(* PLC project PhysicsSimulator, Nammo OpenPLC 1 *)
(* stored: creationDateTime 2026-02-23T12:09:45, modificationDateTime 2026-02-23T12:09:45 *)

TYPE TANK_T : STRUCT
  tank_id : INT;
  status : INT;
  x_position : REAL;
  y_position : REAL;
  z_position : REAL;
  stn_type : INT;
END_STRUCT;
END_TYPE

TYPE STATION_T : STRUCT
  tank_id : INT;
  status : INT;
  x_position : REAL;
  y_position : REAL;
  z_position : REAL;
  stn_type : INT;
  dropping_time : REAL;
  device_delay : REAL;
END_STRUCT;
END_TYPE

TYPE PHYSICS_2D_T : STRUCT
  x_accel_s : REAL;
  x_decel_s : REAL;
  x_max_mm_s : REAL;
  z_total_mm : REAL;
  z_slow_dry_mm : REAL;
  z_slow_wet_mm : REAL;
  z_slow_end_mm : REAL;
  z_slow_mm_s : REAL;
  z_fast_mm_s : REAL;
  drip_delay_s : REAL;
  avoid_mm : REAL;
END_STRUCT;
END_TYPE

TYPE TASK_AREA_T : STRUCT
  min_lift : INT;
  max_lift : INT;
  min_sink : INT;
  max_sink : INT;
END_STRUCT;
END_TYPE

TYPE TRANSPORTER_CFG_T : STRUCT
  x_min_limit : REAL;
  x_max_limit : REAL;
  y_min_limit : REAL;
  y_max_limit : REAL;
  x_avoid_mm : REAL;
  y_avoid_mm : REAL;
  phys2d : PHYSICS_2D_T;
  task_area : ARRAY[1..4] OF TASK_AREA_T;
END_STRUCT;
END_TYPE

TYPE TRANSPORTER_STATE_T : STRUCT
  active : BOOL;
  phase : INT;
  z_stage : INT;
  x_mm : REAL;
  z_mm : REAL;
  vel_x : REAL;
  vel_z : REAL;
  current_station : INT;
  lift_station_target : INT;
  sink_station_target : INT;
  target_x : REAL;
  x_min_limit : REAL;
  x_max_limit : REAL;
  z_timer_s : REAL;
END_STRUCT;
END_TYPE

TYPE BATCH_T : STRUCT
  batch_code : INT;
  state : INT;
  prog_id : INT;
  cur_stage : INT;
END_STRUCT;
END_TYPE

TYPE PROGRAM_STAGE_T : STRUCT
  stations : ARRAY[1..5] OF INT;
  min_time : INT;
  max_time : INT;
  cal_time : INT;
END_STRUCT;
END_TYPE

TYPE TREATMENT_PROGRAM_T : STRUCT
  program_id : INT;
  stages : ARRAY[1..30] OF PROGRAM_STAGE_T;
END_STRUCT;
END_TYPE

TYPE UNIT_T : STRUCT
  location : INT;
  status : INT;
  state : INT;
  target : INT;
END_STRUCT;
END_TYPE

TYPE TSK_STAGE_T : STRUCT
  station : INT;
  entry_time : REAL;
  exit_time : REAL;
  min_time : REAL;
  calc_time : REAL;
  max_time : REAL;
  transfer_time : REAL;
END_STRUCT;
END_TYPE

TYPE TSK_SCHEDULE_T : STRUCT
  stage_count : INT;
  stages : ARRAY[1..30] OF TSK_STAGE_T;
END_STRUCT;
END_TYPE

TYPE TSK_TASK_T : STRUCT
  unit : INT;
  stage : INT;
  lift_station : INT;
  sink_station : INT;
  start_time : REAL;
  finish_time : REAL;
  calc_time : REAL;
  min_time : REAL;
  max_time : REAL;
END_STRUCT;
END_TYPE

TYPE TSK_QUEUE_T : STRUCT
  count : INT;
  queue : ARRAY[1..10] OF TSK_TASK_T;
END_STRUCT;
END_TYPE

TYPE TSK_CHECKED_T : STRUCT
  unit : INT;
  stage : INT;
  transporter : INT;
  start_time : REAL;
  end_time : REAL;
  flex_down : REAL;
  flex_up : REAL;
  x_min : REAL;
  x_max : REAL;
  is_conflict : BOOL;
END_STRUCT;
END_TYPE

TYPE TRAVEL_FROM_T : STRUCT
  to_s : ARRAY[1..25] OF REAL;
END_STRUCT;
END_TYPE

TYPE MOVE_TIMES_T : STRUCT
  lift_s : ARRAY[1..25] OF REAL;
  sink_s : ARRAY[1..25] OF REAL;
  travel : ARRAY[1..25] OF TRAVEL_FROM_T;
END_STRUCT;
END_TYPE

TYPE DEP_IDLE_SLOT_T : STRUCT
  start_time : REAL;
  end_time : REAL;
  lift_station : INT;
  sink_station : INT;
END_STRUCT;
END_TYPE

TYPE DEP_IDLE_SLOT_SET_T : STRUCT
  slots : ARRAY[1..20] OF DEP_IDLE_SLOT_T;
  count : INT;
END_STRUCT;
END_TYPE

TYPE DEP_FIT_RESULT_T : STRUCT
  fits : BOOL;
  delay_s : REAL;
  need_extra_s : REAL;
  task_end_s : REAL;
  slot_idx : INT;
  trans_id : INT;
END_STRUCT;
END_TYPE

TYPE DEP_DELAY_ACTION_T : STRUCT
  stage : INT;
  delay_s : REAL;
  target : INT;
  valid : BOOL;
END_STRUCT;
END_TYPE

TYPE DEP_OVERLAP_T : STRUCT
  flags : ARRAY[101..125] OF BOOL;
  count : INT;
END_STRUCT;
END_TYPE

TYPE DEP_SANDBOX_T : STRUCT
  schedule : ARRAY[1..10] OF TSK_SCHEDULE_T;
  batches : ARRAY[1..10] OF BATCH_T;
  programs : ARRAY[1..10] OF TREATMENT_PROGRAM_T;
  tasks : ARRAY[1..3] OF TSK_QUEUE_T;
  valid : BOOL;
END_STRUCT;
END_TYPE

TYPE DEP_PENDING_WRITE_T : STRUCT
  valid : BOOL;
  programs : ARRAY[1..10] OF TREATMENT_PROGRAM_T;
  schedule : ARRAY[1..10] OF TSK_SCHEDULE_T;
  batch_unit : INT;
  batch_stage : INT;
  time_s : REAL;
END_STRUCT;
END_TYPE

FUNCTION TWA_CalcPriority : REAL
  VAR_INPUT
    i_phase : INT;
    i_can_evade : BOOL;
    i_x_pos : REAL;
    i_x_target : REAL;
  END_VAR
  VAR
    dist : REAL;
  END_VAR

            IF NOT i_can_evade THEN
  TWA_CalcPriority := 100000.0;
  RETURN;
END_IF;

IF i_phase = 3 THEN
  dist := ABS(i_x_pos - i_x_target);
  IF dist > 99999.0 THEN dist := 99999.0; END_IF;
  TWA_CalcPriority := 200000.0 + (99999.0 - dist);
ELSIF i_phase = 1 THEN
  dist := ABS(i_x_pos - i_x_target);
  IF dist > 99999.0 THEN dist := 99999.0; END_IF;
  TWA_CalcPriority := 100000.0 + (99999.0 - dist);
ELSE
  TWA_CalcPriority := 1.0;
END_IF;
          
END_FUNCTION

FUNCTION_BLOCK DEP_FB_CalcIdleSlots
  VAR_INPUT
    i_trans : INT;
    i_time_s : REAL;
  END_VAR
  VAR_EXTERNAL
    g_tasks : ARRAY[1..3] OF TSK_QUEUE_T;
    g_dep_idle_slots : ARRAY[1..3] OF DEP_IDLE_SLOT_SET_T;
  END_VAR
  VAR
    qi : INT;
    si : INT;
    cnt : INT;
    prev_end : REAL;
    prev_sink : INT;
    gap_start : REAL;
    gap_end : REAL;
    HORIZON : REAL := 1.0E9;
  END_VAR

            (* Guard *)
IF i_trans < 1 OR i_trans > 3 THEN
  RETURN;
END_IF;

(* Reset output *)
g_dep_idle_slots[i_trans].count := 0;
si := 0;
cnt := g_tasks[i_trans].count;

prev_end  := i_time_s;
prev_sink := 0;

FOR qi := 1 TO 10 DO
  IF qi > cnt THEN
    EXIT;
  END_IF;

  gap_start := prev_end;
  gap_end   := g_tasks[i_trans].queue[qi].start_time;

  (* Only create slot if there is a meaningful gap *)
  IF gap_end > gap_start + 0.1 THEN
    si := si + 1;
    IF si <= 20 THEN
      g_dep_idle_slots[i_trans].slots[si].start_time   := gap_start;
      g_dep_idle_slots[i_trans].slots[si].end_time     := gap_end;
      g_dep_idle_slots[i_trans].slots[si].lift_station := prev_sink;
      g_dep_idle_slots[i_trans].slots[si].sink_station := g_tasks[i_trans].queue[qi].lift_station;
    END_IF;
  END_IF;

  prev_end  := g_tasks[i_trans].queue[qi].finish_time;
  prev_sink := g_tasks[i_trans].queue[qi].sink_station;
END_FOR;

(* Final slot: after last task → open-ended *)
si := si + 1;
IF si <= 20 THEN
  g_dep_idle_slots[i_trans].slots[si].start_time   := prev_end;
  g_dep_idle_slots[i_trans].slots[si].end_time     := HORIZON;
  g_dep_idle_slots[i_trans].slots[si].lift_station := prev_sink;
  g_dep_idle_slots[i_trans].slots[si].sink_station := 0;
END_IF;

g_dep_idle_slots[i_trans].count := si;
          
END_FUNCTION_BLOCK

FUNCTION_BLOCK DEP_FB_CalcOverlap
  VAR_EXTERNAL
    g_cfg : ARRAY[1..3] OF TRANSPORTER_CFG_T;
    g_dep_overlap : DEP_OVERLAP_T;
  END_VAR
  VAR
    stn : INT;
    ti : INT;
    ai : INT;
    cover_count : INT;
    covered : BOOL;
    area : TASK_AREA_T;
  END_VAR

            g_dep_overlap.count := 0;

FOR stn := 101 TO 125 DO
  cover_count := 0;

  FOR ti := 1 TO 3 DO
    covered := FALSE;
    FOR ai := 1 TO 4 DO
      IF NOT covered THEN
        area := g_cfg[ti].task_area[ai];
        (* Station is covered if within lift OR sink range *)
        IF (area.min_lift > 0 AND stn >= area.min_lift AND stn <= area.max_lift)
           OR (area.min_sink > 0 AND stn >= area.min_sink AND stn <= area.max_sink) THEN
          covered := TRUE;
        END_IF;
      END_IF;
    END_FOR;
    IF covered THEN
      cover_count := cover_count + 1;
    END_IF;
  END_FOR;

  IF cover_count >= 2 THEN
    g_dep_overlap.flags[stn] := TRUE;
    g_dep_overlap.count := g_dep_overlap.count + 1;
  ELSE
    g_dep_overlap.flags[stn] := FALSE;
  END_IF;
END_FOR;
          
END_FUNCTION_BLOCK

FUNCTION_BLOCK STC_FB_CalcHorizontalTravel
  VAR_INPUT
    i_from_stn : INT;
    i_to_stn : INT;
    i_trans : INT;
  END_VAR
  VAR_OUTPUT
    o_travel_s : REAL;
  END_VAR
  VAR_EXTERNAL
    g_move : ARRAY[1..3] OF MOVE_TIMES_T;
  END_VAR
  VAR
    from_idx : INT;
    to_idx : INT;
  END_VAR

            o_travel_s := 0.0;
IF i_from_stn > 0 AND i_to_stn > 0 AND i_from_stn <> i_to_stn THEN
  from_idx := i_from_stn - 100;
  to_idx   := i_to_stn - 100;
  IF from_idx >= 1 AND from_idx <= 25 AND to_idx >= 1 AND to_idx <= 25
     AND i_trans >= 1 AND i_trans <= 3 THEN
    o_travel_s := g_move[i_trans].travel[from_idx].to_s[to_idx];
  END_IF;
END_IF;
          
END_FUNCTION_BLOCK

FUNCTION_BLOCK DEP_FB_FitTaskToSlot
  VAR_INPUT
    i_lift_stn : INT;
    i_sink_stn : INT;
    i_trans_id : INT;
    i_task_start : REAL;
    i_task_end : REAL;
    i_shift_s : REAL;
    i_calc_time_s : REAL;
    i_max_time_s : REAL;
    i_flex_factor : REAL;
    i_margin_s : REAL;
  END_VAR
  VAR_OUTPUT
    o_result : DEP_FIT_RESULT_T;
  END_VAR
  VAR_EXTERNAL
    g_dep_idle_slots : ARRAY[1..3] OF DEP_IDLE_SLOT_SET_T;
  END_VAR
  VAR
    fb_travel_to : STC_FB_CalcHorizontalTravel;
    fb_travel_from : STC_FB_CalcHorizontalTravel;
    si : INT;
    slot_cnt : INT;
    slot_start : REAL;
    slot_end : REAL;
    from_stn : INT;
    to_stn : INT;
    travel_to : REAL;
    travel_from : REAL;
    earliest : REAL;
    latest : REAL;
    task_dur : REAL;
    delay : REAL;
    flex_up : REAL;
    capped_flex : REAL;
    best_delay : REAL;
    best_slot : INT;
    found : BOOL;
  END_VAR

            (* Initialize output *)
o_result.fits         := FALSE;
o_result.delay_s      := 0.0;
o_result.need_extra_s := 0.0;
o_result.task_end_s   := 0.0;
o_result.slot_idx     := 0;
o_result.trans_id     := i_trans_id;

IF i_trans_id < 1 OR i_trans_id > 3 THEN
  RETURN;
END_IF;

task_dur   := i_task_end - i_task_start;
flex_up    := i_max_time_s - i_calc_time_s;
IF flex_up < 0.0 THEN flex_up := 0.0; END_IF;
capped_flex := flex_up * i_flex_factor;

slot_cnt   := g_dep_idle_slots[i_trans_id].count;
best_delay := 1.0E9;
best_slot  := 0;
found      := FALSE;

FOR si := 1 TO 20 DO
  IF si > slot_cnt THEN
    EXIT;
  END_IF;

  slot_start := g_dep_idle_slots[i_trans_id].slots[si].start_time;
  slot_end   := g_dep_idle_slots[i_trans_id].slots[si].end_time;

  (* ── Travel time: prev task sink → this lift ── *)
  from_stn := g_dep_idle_slots[i_trans_id].slots[si].lift_station;
  travel_to := 0.0;
  IF from_stn > 0 AND from_stn <> i_lift_stn THEN
    fb_travel_to(i_from_stn := from_stn, i_to_stn := i_lift_stn, i_trans := i_trans_id);
    travel_to := fb_travel_to.o_travel_s;
  END_IF;

  (* ── Travel time: this sink → next task lift ── *)
  to_stn := g_dep_idle_slots[i_trans_id].slots[si].sink_station;
  travel_from := 0.0;
  IF to_stn > 0 AND to_stn <> i_sink_stn THEN
    fb_travel_from(i_from_stn := i_sink_stn, i_to_stn := to_stn, i_trans := i_trans_id);
    travel_from := fb_travel_from.o_travel_s;
  END_IF;

  (* Earliest start = max(slot_start, task_start + shift) + travel_to + margin *)
  IF slot_start > (i_task_start + i_shift_s) THEN
    earliest := slot_start + travel_to + i_margin_s;
  ELSE
    earliest := i_task_start + i_shift_s + travel_to + i_margin_s;
  END_IF;

  (* Latest end = slot_end - travel_from - margin *)
  IF slot_end > 1.0E8 THEN
    (* Open-ended slot *)
    latest := 1.0E8;
  ELSE
    latest := slot_end - travel_from - i_margin_s;
  END_IF;

  (* Check if task fits *)
  IF earliest + task_dur <= latest THEN
    delay := earliest - i_task_start - i_shift_s;
    IF delay < 0.0 THEN delay := 0.0; END_IF;

    (* Flex constraint: delay must not exceed capped flex *)
    IF delay <= capped_flex + i_margin_s THEN
      IF delay < best_delay THEN
        best_delay := delay;
        best_slot  := si;
        found      := TRUE;
      END_IF;
    END_IF;
  END_IF;
END_FOR;

IF found THEN
  o_result.fits      := TRUE;
  o_result.delay_s   := best_delay;
  o_result.slot_idx  := best_slot;
  o_result.task_end_s := i_task_start + i_shift_s + best_delay + task_dur;
  o_result.need_extra_s := 0.0;
ELSE
  (* Report how much extra is needed for backward chaining *)
  (* Use the best near-miss: smallest overshoot beyond capped_flex *)
  o_result.fits := FALSE;
  IF best_delay < 1.0E8 THEN
    o_result.need_extra_s := best_delay - capped_flex;
    IF o_result.need_extra_s < 0.0 THEN
      o_result.need_extra_s := 0.0;
    END_IF;
  ELSE
    o_result.need_extra_s := 0.0;  (* no slot at all *)
  END_IF;
END_IF;
          
END_FUNCTION_BLOCK

FUNCTION_BLOCK DEP_FB_OverlapDelay
  VAR_INPUT
    i_lift_stn : INT;
    i_sink_stn : INT;
    i_trans_id : INT;
    i_task_start : REAL;
    i_task_end : REAL;
    i_margin_s : REAL;
  END_VAR
  VAR_OUTPUT
    o_delay_s : REAL;
  END_VAR
  VAR_EXTERNAL
    g_tasks : ARRAY[1..3] OF TSK_QUEUE_T;
    g_dep_overlap : DEP_OVERLAP_T;
  END_VAR
  VAR
    lift_is_overlap : BOOL;
    sink_is_overlap : BOOL;
    round : INT;
    ti : INT;
    qi : INT;
    max_conf : REAL;
    t_start : REAL;
    t_end : REAL;
    e_start : REAL;
    e_end : REAL;
    e_lift : INT;
    e_sink : INT;
    has_ovlp : BOOL;
    needed : REAL;
  END_VAR

            o_delay_s := 0.0;

(* Check if lift/sink are in overlap zone *)
IF i_lift_stn >= 101 AND i_lift_stn <= 125 THEN
  lift_is_overlap := g_dep_overlap.flags[i_lift_stn];
ELSE
  lift_is_overlap := FALSE;
END_IF;
IF i_sink_stn >= 101 AND i_sink_stn <= 125 THEN
  sink_is_overlap := g_dep_overlap.flags[i_sink_stn];
ELSE
  sink_is_overlap := FALSE;
END_IF;

(* No overlap stations involved → no delay *)
IF NOT lift_is_overlap AND NOT sink_is_overlap THEN
  RETURN;
END_IF;

(* Iterative conflict resolution — max 20 rounds *)
FOR round := 1 TO 20 DO
  max_conf := 0.0;
  t_start  := i_task_start + o_delay_s;
  t_end    := i_task_end + o_delay_s;

  (* Check all tasks on OTHER transporters *)
  FOR ti := 1 TO 3 DO
    IF ti <> i_trans_id THEN
      FOR qi := 1 TO 10 DO
        IF qi > g_tasks[ti].count THEN
          EXIT;
        END_IF;

        e_lift  := g_tasks[ti].queue[qi].lift_station;
        e_sink  := g_tasks[ti].queue[qi].sink_station;
        e_start := g_tasks[ti].queue[qi].start_time;
        e_end   := g_tasks[ti].queue[qi].finish_time;

        (* Does existing task share an overlap station? *)
        has_ovlp := FALSE;
        IF lift_is_overlap AND (e_lift = i_lift_stn OR e_sink = i_lift_stn) THEN
          has_ovlp := TRUE;
        END_IF;
        IF sink_is_overlap AND (e_lift = i_sink_stn OR e_sink = i_sink_stn) THEN
          has_ovlp := TRUE;
        END_IF;

        IF has_ovlp THEN
          (* Time overlap check: task overlaps with existing? *)
          IF t_start < (e_end + i_margin_s) AND t_end > (e_start - i_margin_s) THEN
            needed := (e_end + i_margin_s) - t_start;
            IF needed > max_conf THEN
              max_conf := needed;
            END_IF;
          END_IF;
        END_IF;

      END_FOR;  (* qi *)
    END_IF;
  END_FOR;  (* ti *)

  (* No conflict found → done *)
  IF max_conf <= 0.0 THEN
    EXIT;
  END_IF;
  o_delay_s := o_delay_s + max_conf;
END_FOR;  (* round *)
          
END_FUNCTION_BLOCK

FUNCTION_BLOCK DEP_FB_Sandbox
  VAR_INPUT
    i_cmd : INT;
  END_VAR
  VAR_EXTERNAL
    g_schedule : ARRAY[1..10] OF TSK_SCHEDULE_T;
    g_batches : ARRAY[1..10] OF BATCH_T;
    g_programs : ARRAY[1..10] OF TREATMENT_PROGRAM_T;
    g_tasks : ARRAY[1..3] OF TSK_QUEUE_T;
    g_dep_sandbox : DEP_SANDBOX_T;
  END_VAR
  VAR
    ui : INT;
    ti : INT;
  END_VAR

            IF i_cmd = 1 THEN
  (* ── SNAPSHOT: globals → sandbox ── *)
  FOR ui := 1 TO 10 DO
    g_dep_sandbox.schedule[ui] := g_schedule[ui];
    g_dep_sandbox.batches[ui]  := g_batches[ui];
    g_dep_sandbox.programs[ui] := g_programs[ui];
  END_FOR;
  FOR ti := 1 TO 3 DO
    g_dep_sandbox.tasks[ti] := g_tasks[ti];
  END_FOR;
  g_dep_sandbox.valid := TRUE;

ELSIF i_cmd = 2 THEN
  (* ── RESTORE: sandbox → globals ── *)
  IF g_dep_sandbox.valid THEN
    FOR ui := 1 TO 10 DO
      g_schedule[ui] := g_dep_sandbox.schedule[ui];
      g_batches[ui]  := g_dep_sandbox.batches[ui];
      g_programs[ui] := g_dep_sandbox.programs[ui];
    END_FOR;
    FOR ti := 1 TO 3 DO
      g_tasks[ti] := g_dep_sandbox.tasks[ti];
    END_FOR;
  END_IF;

ELSIF i_cmd = 3 THEN
  (* ── CLEAR: invalidate sandbox ── *)
  g_dep_sandbox.valid := FALSE;

END_IF;
          
END_FUNCTION_BLOCK

FUNCTION_BLOCK STC_FB_CalcTransferTime
  VAR_INPUT
    i_from_stn : INT;
    i_to_stn : INT;
    i_trans : INT;
  END_VAR
  VAR_OUTPUT
    o_total_s : REAL;
    o_lift_s : REAL;
    o_travel_s : REAL;
    o_sink_s : REAL;
  END_VAR
  VAR_EXTERNAL
    g_move : ARRAY[1..3] OF MOVE_TIMES_T;
  END_VAR
  VAR
    from_idx : INT;
    to_idx : INT;
  END_VAR

            o_total_s  := 0.0;
o_lift_s   := 0.0;
o_travel_s := 0.0;
o_sink_s   := 0.0;

IF i_from_stn > 0 AND i_from_stn <> i_to_stn THEN
  from_idx := i_from_stn - 100;
  to_idx   := i_to_stn - 100;
  IF from_idx >= 1 AND from_idx <= 25 AND to_idx >= 1 AND to_idx <= 25
     AND i_trans >= 1 AND i_trans <= 3 THEN
    o_lift_s   := g_move[i_trans].lift_s[from_idx];
    o_travel_s := g_move[i_trans].travel[from_idx].to_s[to_idx];
    o_sink_s   := g_move[i_trans].sink_s[to_idx];
    o_total_s  := o_lift_s + o_travel_s + o_sink_s;
  END_IF;
END_IF;
          
END_FUNCTION_BLOCK

FUNCTION_BLOCK STC_FB_FindTransporter
  VAR_INPUT
    i_lift_stn : INT;
    i_sink_stn : INT;
  END_VAR
  VAR_OUTPUT
    o_trans_id : INT;
  END_VAR
  VAR_EXTERNAL
    g_cfg : ARRAY[1..3] OF TRANSPORTER_CFG_T;
  END_VAR
  VAR
    ti : INT;
    ai : INT;
    area : TASK_AREA_T;
    can_lift : BOOL;
    can_sink : BOOL;
  END_VAR

            o_trans_id := 0;
FOR ti := 1 TO 3 DO
  IF o_trans_id = 0 THEN
    FOR ai := 1 TO 4 DO
      IF o_trans_id = 0 THEN
        area := g_cfg[ti].task_area[ai];
        IF area.min_lift > 0 OR area.max_lift > 0 THEN
          can_lift := (i_lift_stn >= area.min_lift) AND (i_lift_stn <= area.max_lift);
          IF i_sink_stn = 0 THEN
            (* Lift-only coverage search *)
            IF can_lift THEN
              o_trans_id := ti;
            END_IF;
          ELSE
            can_sink := (i_sink_stn >= area.min_sink) AND (i_sink_stn <= area.max_sink);
            IF can_lift AND can_sink THEN
              o_trans_id := ti;
            END_IF;
          END_IF;
        END_IF;
      END_IF;
    END_FOR;
  END_IF;
END_FOR;
          
END_FUNCTION_BLOCK

FUNCTION_BLOCK TSK_FB_CalcSchedule
  VAR_INPUT
    i_unit : INT;
    i_trans : INT;
    i_time_s : REAL;
  END_VAR
  VAR_EXTERNAL
    g_batches : ARRAY[1..10] OF BATCH_T;
    g_programs : ARRAY[1..10] OF TREATMENT_PROGRAM_T;
    g_units : ARRAY[1..10] OF UNIT_T;
    g_stations : ARRAY[101..125] OF STATION_T;
    g_schedule : ARRAY[1..10] OF TSK_SCHEDULE_T;
    g_station_count : INT;
  END_VAR
  VAR
    st : INT;
    stn_num : INT;
    prev_stn : INT;
    cur_stage : INT;
    location : INT;
    start_st : INT;
    entry_t : REAL;
    exit_t : REAL;
    xfer_t : REAL;
    calc_s : REAL;
    min_s : REAL;
    max_s : REAL;
    is_on_stn : BOOL;
    is_first : BOOL;
    remain_s : REAL;
    elapsed_s : REAL;
    out_count : INT;
    p : INT;
    chosen_stn : INT;
    fb_xfer : STC_FB_CalcTransferTime;
  END_VAR

            (* -- Validate inputs -- *)
IF i_unit < 1 OR i_unit > 10 THEN RETURN; END_IF;
IF i_trans < 1 OR i_trans > 3 THEN RETURN; END_IF;

(* -- Read batch and unit data -- *)
cur_stage := g_batches[i_unit].cur_stage;
location  := g_units[i_unit].location;
is_on_stn := location >= 100;
out_count := 0;

(* -- Clear old schedule -- *)
FOR st := 1 TO 30 DO
  g_schedule[i_unit].stages[st].station := 0;
  g_schedule[i_unit].stages[st].entry_time := 0.0;
  g_schedule[i_unit].stages[st].exit_time := 0.0;
  g_schedule[i_unit].stages[st].min_time := 0.0;
  g_schedule[i_unit].stages[st].calc_time := 0.0;
  g_schedule[i_unit].stages[st].max_time := 0.0;
  g_schedule[i_unit].stages[st].transfer_time := 0.0;
END_FOR;

(* -- Determine start stage -- *)
(* Stage 90 = waiting batch, treat as stage 0 *)
IF cur_stage = 90 THEN
  cur_stage := 0;
END_IF;

(* If on transporter, start from next stage; if on station, from current *)
IF is_on_stn THEN
  start_st := cur_stage;
ELSE
  start_st := cur_stage + 1;
END_IF;

(* Force minimum stage 1 *)
IF start_st < 1 THEN
  start_st := 1;
END_IF;

(* -- Previous station (where transfer starts from) -- *)
IF is_on_stn THEN
  prev_stn := location;
ELSIF cur_stage >= 1 AND cur_stage <= 30 THEN
  (* On transporter: use previous stage station *)
  prev_stn := g_programs[i_unit].stages[cur_stage].stations[1];
ELSE
  prev_stn := 0;
END_IF;

(* -- prevExitTime: when next stage can begin -- *)
IF is_on_stn THEN
  (* Unit is on station: calculate remaining time *)
  calc_s := INT_TO_REAL(g_batches[i_unit].cur_stage);
  (* For first stage, remaining time based on calc_time *)
  exit_t := i_time_s;
ELSE
  exit_t := i_time_s;
END_IF;

is_first := TRUE;

(* ============================================================
   MAIN LOOP: Calculate schedule for each program stage
   ============================================================ *)
FOR st := start_st TO 30 DO

  (* Check if stage has a valid station *)
  chosen_stn := 0;
  FOR p := 1 TO 5 DO
    IF g_programs[i_unit].stages[st].stations[p] > 0 AND chosen_stn = 0 THEN
      chosen_stn := g_programs[i_unit].stages[st].stations[p];
    END_IF;
  END_FOR;

  (* No station means end of program *)
  IF chosen_stn = 0 THEN
    EXIT;
  END_IF;

  stn_num := chosen_stn;

  (* Read treatment times from program *)
  calc_s := INT_TO_REAL(g_programs[i_unit].stages[st].cal_time);
  min_s  := INT_TO_REAL(g_programs[i_unit].stages[st].min_time);
  max_s  := INT_TO_REAL(g_programs[i_unit].stages[st].max_time);

  (* -- Calculate transfer time from prev_stn to stn_num -- *)
  fb_xfer(i_from_stn := prev_stn, i_to_stn := stn_num, i_trans := i_trans);
  xfer_t := fb_xfer.o_total_s;

  (* -- Calculate entry and exit times -- *)
  IF is_first AND is_on_stn AND st = cur_stage THEN
    (* Batch is currently at this station *)
    entry_t := i_time_s;
    (* Remaining time: calc_time - elapsed *)
    remain_s := calc_s;
    IF remain_s < 1.0 THEN remain_s := 1.0; END_IF;
    exit_t := i_time_s + remain_s;
  ELSIF is_first AND NOT is_on_stn THEN
    (* Batch is on transporter: entry = now (transfer in progress) *)
    entry_t := exit_t;
    exit_t  := entry_t + calc_s;
  ELSE
    (* Normal stage: entry = prev exit + transfer *)
    entry_t := exit_t + xfer_t;
    exit_t  := entry_t + calc_s;
  END_IF;

  (* -- Write to schedule -- *)
  out_count := out_count + 1;
  IF out_count <= 30 THEN
    g_schedule[i_unit].stages[out_count].station       := stn_num;
    g_schedule[i_unit].stages[out_count].entry_time    := entry_t;
    g_schedule[i_unit].stages[out_count].exit_time     := exit_t;
    g_schedule[i_unit].stages[out_count].min_time      := min_s;
    g_schedule[i_unit].stages[out_count].calc_time     := calc_s;
    g_schedule[i_unit].stages[out_count].max_time      := max_s;
    g_schedule[i_unit].stages[out_count].transfer_time := xfer_t;
  END_IF;

  (* -- Update for next iteration -- *)
  prev_stn := stn_num;
  is_first := FALSE;

END_FOR;

g_schedule[i_unit].stage_count := out_count;
          
END_FUNCTION_BLOCK

FUNCTION_BLOCK TSK_FB_CreateTasks
  VAR_INPUT
    i_unit : INT;
  END_VAR
  VAR_EXTERNAL
    g_batches : ARRAY[1..10] OF BATCH_T;
    g_schedule : ARRAY[1..10] OF TSK_SCHEDULE_T;
    g_tasks : ARRAY[1..3] OF TSK_QUEUE_T;
  END_VAR
  VAR
    si : INT;
    sc : INT;
    lift_stn : INT;
    sink_stn : INT;
    cur_stage : INT;
    skip_before : INT;
    tid : INT;
    qi : INT;
    stg_num : INT;
    fb_find : STC_FB_FindTransporter;
  END_VAR

            IF i_unit < 1 OR i_unit > 10 THEN RETURN; END_IF;

sc := g_schedule[i_unit].stage_count;
IF sc < 2 THEN RETURN; END_IF;

cur_stage := g_batches[i_unit].cur_stage;
IF cur_stage = 90 THEN
  skip_before := 0;
ELSE
  skip_before := cur_stage;
END_IF;

(* Loop through consecutive stage pairs *)
FOR si := 1 TO sc - 1 DO
  (* schedule index si = current stage, si+1 = next stage *)
  stg_num := si;   (* simplified: schedule stage index = stage number *)

  (* Skip already completed stages *)
  IF stg_num >= skip_before THEN
    lift_stn := g_schedule[i_unit].stages[si].station;
    sink_stn := g_schedule[i_unit].stages[si + 1].station;

    IF lift_stn > 0 AND sink_stn > 0 THEN
      (* -- Find transporter via task_area matching -- *)
      fb_find(i_lift_stn := lift_stn, i_sink_stn := sink_stn);
      tid := fb_find.o_trans_id;

      (* -- Append task to transporter queue -- *)
      IF tid >= 1 AND tid <= 3 THEN
        qi := g_tasks[tid].count + 1;
        IF qi <= 10 THEN
          g_tasks[tid].queue[qi].unit         := i_unit;
          g_tasks[tid].queue[qi].stage        := stg_num;
          g_tasks[tid].queue[qi].lift_station := lift_stn;
          g_tasks[tid].queue[qi].sink_station := sink_stn;
          g_tasks[tid].queue[qi].start_time   := g_schedule[i_unit].stages[si].exit_time;
          g_tasks[tid].queue[qi].finish_time  := g_schedule[i_unit].stages[si + 1].entry_time;
          g_tasks[tid].queue[qi].calc_time    := g_schedule[i_unit].stages[si].calc_time;
          g_tasks[tid].queue[qi].min_time     := g_schedule[i_unit].stages[si].min_time;
          g_tasks[tid].queue[qi].max_time     := g_schedule[i_unit].stages[si].max_time;
          g_tasks[tid].count := qi;
        END_IF;
      END_IF;
    END_IF;
  END_IF;
END_FOR;
          
END_FUNCTION_BLOCK

FUNCTION_BLOCK TSK_FB_SwapTasks
  VAR_OUTPUT
    o_swap_count : INT;
  END_VAR
  VAR_EXTERNAL
    g_tasks : ARRAY[1..3] OF TSK_QUEUE_T;
  END_VAR
  VAR
    ti : INT;
    qi : INT;
    cnt : INT;
    tmp : TSK_TASK_T;
  END_VAR

            o_swap_count := 0;

FOR ti := 1 TO 3 DO
  cnt := g_tasks[ti].count;
  IF cnt >= 2 THEN
    FOR qi := 1 TO cnt - 1 DO
      (* Check: different units AND prev.sink == next.lift *)
      IF g_tasks[ti].queue[qi].unit <> g_tasks[ti].queue[qi + 1].unit
         AND g_tasks[ti].queue[qi].sink_station = g_tasks[ti].queue[qi + 1].lift_station THEN
        (* Swap *)
        tmp := g_tasks[ti].queue[qi];
        g_tasks[ti].queue[qi] := g_tasks[ti].queue[qi + 1];
        g_tasks[ti].queue[qi + 1] := tmp;
        o_swap_count := o_swap_count + 1;
      END_IF;
    END_FOR;
  END_IF;
END_FOR;
          
END_FUNCTION_BLOCK

FUNCTION_BLOCK DEP_FB_Scheduler
  VAR_INPUT
    i_run : BOOL;
    i_time_s : REAL;
    i_tsk_phase : INT;
  END_VAR
  VAR_OUTPUT
    o_phase : INT;
    o_wait_cnt : INT;
    o_activated : BOOL;
  END_VAR
  VAR_EXTERNAL
    g_batches : ARRAY[1..10] OF BATCH_T;
    g_units : ARRAY[1..10] OF UNIT_T;
    g_programs : ARRAY[1..10] OF TREATMENT_PROGRAM_T;
    g_schedule : ARRAY[1..10] OF TSK_SCHEDULE_T;
    g_tasks : ARRAY[1..3] OF TSK_QUEUE_T;
    g_cfg : ARRAY[1..3] OF TRANSPORTER_CFG_T;
    g_dep_sandbox : DEP_SANDBOX_T;
    g_dep_idle_slots : ARRAY[1..3] OF DEP_IDLE_SLOT_SET_T;
    g_dep_overlap : DEP_OVERLAP_T;
    g_dep_pending : DEP_PENDING_WRITE_T;
    g_dep_activated : BOOL;
    g_dep_stable : BOOL;
    g_dep_waiting : ARRAY[1..10] OF INT;
    g_dep_waiting_count : INT;
  END_VAR
  VAR
    phase : INT := 0;
    next_phase : INT;
    waiting_list : ARRAY[1..10] OF INT;
    waiting_cnt : INT;
    cur_wait_idx : INT;
    cur_wait_unit : INT;
    batch_list : ARRAY[1..10] OF INT;
    batch_count : INT;
    w_tasks : ARRAY[1..30] OF TSK_TASK_T;
    w_trans : ARRAY[1..30] OF INT;
    w_task_cnt : INT;
    cur_task_idx : INT;
    fit_round : INT;
    MAX_FIT_ROUNDS : INT := 50;
    sched_base_time : REAL;
    delay_stage : INT;
    delay_amount : REAL;
    delay_target : INT;
    FLEX_FACTOR : REAL := 0.5;
    MARGIN_S : REAL := 5.0;
    CONFLICT_MARGIN_S : REAL := 1.0;
    MAX_INIT_WAIT_S : REAL := 120.0;
    END_DELAY_TICKS : INT := 100;
    end_delay_cnt : INT;
    fb_sandbox : DEP_FB_Sandbox;
    fb_overlap : DEP_FB_CalcOverlap;
    fb_idle_slots : DEP_FB_CalcIdleSlots;
    fb_fit : DEP_FB_FitTaskToSlot;
    fb_ovlp_delay : DEP_FB_OverlapDelay;
    fb_calc_sched : TSK_FB_CalcSchedule;
    fb_create_tasks : TSK_FB_CreateTasks;
    fb_swap_tasks : TSK_FB_SwapTasks;
    fb_find_trans : STC_FB_FindTransporter;
    fb_xfer : STC_FB_CalcTransferTime;
    ti : INT;
    sched_trans : INT;
    write_idx : INT;
    loading_stn : INT;
    first_stn : INT;
    xfer_dur : REAL;
    stage0_delay : REAL;
    ovlp_delay_s : REAL;
    total_delay_s : REAL;
    prog_idx : INT;
    old_cal : INT;
    new_cal : INT;
    max_cal : INT;
    ins_i : INT;
    ins_j : INT;
    ins_cnt : INT;
    tmp_task : TSK_TASK_T;
  END_VAR

            IF NOT i_run THEN
  phase := 0;
  o_phase := 0;
  o_activated := FALSE;
  RETURN;
END_IF;

next_phase := phase;
o_activated := FALSE;

(* ════════════════════════════════════════════════════════════ *)
(* PHASE 0: STOPPED                                           *)
(* ════════════════════════════════════════════════════════════ *)
IF phase = 0 THEN
  next_phase := 1;

(* ════════════════════════════════════════════════════════════ *)
(* PHASE 1: WAIT_STABLE                                       *)
(* Wait for TSK to be ready (phase >= 10000)                   *)
(* ════════════════════════════════════════════════════════════ *)
ELSIF phase = 1 THEN
  IF i_tsk_phase >= 10000 AND g_dep_stable THEN
    next_phase := 100;
  END_IF;

(* ════════════════════════════════════════════════════════════ *)
(* PHASE 100: INIT — snapshot sandbox, find waiting batches    *)
(* ════════════════════════════════════════════════════════════ *)
ELSIF phase = 100 THEN
  (* Snapshot globals → sandbox (backup for rollback) *)
  fb_sandbox(i_cmd := 1);

  (* Find waiting batches (cur_stage = 90) *)
  waiting_cnt := 0;
  FOR ui := 1 TO 10 DO
    IF g_batches[ui].state = 1 AND g_batches[ui].cur_stage = 90 THEN
      (* Check unit target is 'none' (TO_NONE = 0) *)
      IF g_units[ui].target = 0 THEN
        waiting_cnt := waiting_cnt + 1;
        waiting_list[waiting_cnt] := ui;
      END_IF;
    END_IF;
  END_FOR;

  o_wait_cnt := waiting_cnt;
  g_dep_waiting_count := waiting_cnt;
  FOR ui := 1 TO waiting_cnt DO
    g_dep_waiting[ui] := waiting_list[ui];
  END_FOR;

  (* Build active batch list for rebuild phases *)
  batch_count := 0;
  FOR ui := 1 TO 10 DO
    IF g_batches[ui].state = 1 THEN
      batch_count := batch_count + 1;
      batch_list[batch_count] := ui;
    END_IF;
  END_FOR;

  IF waiting_cnt = 0 THEN
    (* No waiting batches → back to waiting *)
    fb_sandbox(i_cmd := 3);   (* clear sandbox *)
    next_phase := 1;
  ELSE
    cur_wait_idx := 1;
    next_phase := 200;
  END_IF;

(* ════════════════════════════════════════════════════════════ *)
(* PHASE 200: CALC_OVERLAP — compute overlap stations          *)
(* ════════════════════════════════════════════════════════════ *)
ELSIF phase = 200 THEN
  fb_overlap();
  next_phase := 1000;

(* ════════════════════════════════════════════════════════════ *)
(* PHASE 1000: BATCH_START — prepare current waiting batch     *)
(* ════════════════════════════════════════════════════════════ *)
ELSIF phase = 1000 THEN
  IF cur_wait_idx > waiting_cnt THEN
    (* All batches processed, none activated → back to waiting *)
    fb_sandbox(i_cmd := 2);   (* restore globals from snapshot *)
    fb_sandbox(i_cmd := 3);   (* clear sandbox *)
    next_phase := 1;
  ELSE
    cur_wait_unit := waiting_list[cur_wait_idx];
    fit_round := 0;
    sched_base_time := i_time_s;
    next_phase := 1010;
  END_IF;

(* ════════════════════════════════════════════════════════════ *)
(* PHASE 1010: CALC_SCHED — calculate waiting batch schedule   *)
(* ════════════════════════════════════════════════════════════ *)
ELSIF phase = 1010 THEN
  (* Find transporter for this batch based on its location *)
  fb_find_trans(i_lift_stn := g_units[cur_wait_unit].location, i_sink_stn := 0);
  sched_trans := fb_find_trans.o_trans_id;
  IF sched_trans = 0 THEN sched_trans := 1; END_IF;

  (* Calculate schedule using (possibly shifted) base time *)
  fb_calc_sched(
    i_unit   := cur_wait_unit,
    i_trans  := sched_trans,
    i_time_s := sched_base_time
  );

  next_phase := 1020;

(* ════════════════════════════════════════════════════════════ *)
(* PHASE 1020: REBUILD_TASKS — rebuild all task queues         *)
(* Clear, create for all active batches, sort, swap — one tick *)
(* ════════════════════════════════════════════════════════════ *)
ELSIF phase = 1020 THEN
  (* Clear all task queues *)
  FOR ti := 1 TO 3 DO
    g_tasks[ti].count := 0;
    FOR qi := 1 TO 10 DO
      g_tasks[ti].queue[qi].unit := 0;
      g_tasks[ti].queue[qi].stage := 0;
      g_tasks[ti].queue[qi].lift_station := 0;
      g_tasks[ti].queue[qi].sink_station := 0;
      g_tasks[ti].queue[qi].start_time := 0.0;
      g_tasks[ti].queue[qi].finish_time := 0.0;
      g_tasks[ti].queue[qi].calc_time := 0.0;
      g_tasks[ti].queue[qi].min_time := 0.0;
      g_tasks[ti].queue[qi].max_time := 0.0;
    END_FOR;
  END_FOR;

  (* Create tasks for ALL active batches *)
  FOR bi := 1 TO batch_count DO
    fb_create_tasks(i_unit := batch_list[bi]);
  END_FOR;

  (* Insertion sort each queue by start_time *)
  FOR ti := 1 TO 3 DO
    ins_cnt := g_tasks[ti].count;
    IF ins_cnt >= 2 THEN
      FOR ins_i := 2 TO ins_cnt DO
        tmp_task := g_tasks[ti].queue[ins_i];
        ins_j := ins_i - 1;
        WHILE ins_j >= 1 AND g_tasks[ti].queue[ins_j].start_time > tmp_task.start_time DO
          g_tasks[ti].queue[ins_j + 1] := g_tasks[ti].queue[ins_j];
          ins_j := ins_j - 1;
        END_WHILE;
        g_tasks[ti].queue[ins_j + 1] := tmp_task;
      END_FOR;
    END_IF;
  END_FOR;

  (* Swap same-station pairs *)
  fb_swap_tasks();

  next_phase := 1030;

(* ════════════════════════════════════════════════════════════ *)
(* PHASE 1030: EXTRACT_WAIT — extract waiting batch tasks      *)
(* Copy waiting batch's tasks to w_tasks[], remove from queues *)
(* ════════════════════════════════════════════════════════════ *)
ELSIF phase = 1030 THEN
  w_task_cnt := 0;

  FOR ti := 1 TO 3 DO
    write_idx := 0;
    FOR qi := 1 TO g_tasks[ti].count DO
      IF g_tasks[ti].queue[qi].unit = cur_wait_unit THEN
        (* Copy to waiting task array *)
        w_task_cnt := w_task_cnt + 1;
        IF w_task_cnt <= 30 THEN
          w_tasks[w_task_cnt] := g_tasks[ti].queue[qi];
          w_trans[w_task_cnt] := ti;
        END_IF;
      ELSE
        (* Keep in queue — shift down *)
        write_idx := write_idx + 1;
        IF write_idx <> qi THEN
          g_tasks[ti].queue[write_idx] := g_tasks[ti].queue[qi];
        END_IF;
      END_IF;
    END_FOR;
    (* Clear remaining slots *)
    FOR qi := write_idx + 1 TO g_tasks[ti].count DO
      g_tasks[ti].queue[qi].unit := 0;
    END_FOR;
    g_tasks[ti].count := write_idx;
  END_FOR;

  next_phase := 1040;

(* ════════════════════════════════════════════════════════════ *)
(* PHASE 1040: CALC_IDLE — calc idle slots for all transporters*)
(* ════════════════════════════════════════════════════════════ *)
ELSIF phase = 1040 THEN
  FOR ti := 1 TO 3 DO
    fb_idle_slots(i_trans := ti, i_time_s := i_time_s);
  END_FOR;
  cur_task_idx := 1;
  next_phase := 2000;

(* ════════════════════════════════════════════════════════════ *)
(* PHASE 2000: FIT_STAGE0 — check pickup from loading station *)
(* Uses DEP_FB_FitTaskToSlot to fit the virtual pickup task    *)
(* ════════════════════════════════════════════════════════════ *)
ELSIF phase = 2000 THEN
  loading_stn := g_units[cur_wait_unit].location;

  (* Find first treatment station from schedule *)
  first_stn := 0;
  IF g_schedule[cur_wait_unit].stage_count >= 1 THEN
    first_stn := g_schedule[cur_wait_unit].stages[1].station;
  END_IF;

  IF first_stn = 0 OR loading_stn < 100 THEN
    (* No valid schedule or batch not on station → reject *)
    next_phase := 9000;
  ELSE
    (* Find transporter for pickup *)
    fb_find_trans(i_lift_stn := loading_stn, i_sink_stn := first_stn);
    sched_trans := fb_find_trans.o_trans_id;
    IF sched_trans = 0 THEN sched_trans := 1; END_IF;

    (* Calculate transfer time for pickup *)
    fb_xfer(i_from_stn := loading_stn, i_to_stn := first_stn, i_trans := sched_trans);
    xfer_dur := fb_xfer.o_total_s;
    IF xfer_dur < 1.0 THEN xfer_dur := 1.0; END_IF;

    (* Try fitting pickup into idle slots *)
    fb_fit(
      i_lift_stn     := loading_stn,
      i_sink_stn     := first_stn,
      i_trans_id     := sched_trans,
      i_task_start   := sched_base_time,
      i_task_end     := sched_base_time + xfer_dur,
      i_shift_s      := 0.0,
      i_calc_time_s  := 0.0,
      i_max_time_s   := 2.0 * MAX_INIT_WAIT_S,
      i_flex_factor  := FLEX_FACTOR,
      i_margin_s     := MARGIN_S
    );

    IF fb_fit.o_result.fits THEN
      stage0_delay := fb_fit.o_result.delay_s;

      IF stage0_delay > MARGIN_S THEN
        (* Stage 0 needs delay — shift base time and recalculate *)
        sched_base_time := sched_base_time + stage0_delay;
        fit_round := fit_round + 1;
        IF fit_round > MAX_FIT_ROUNDS THEN
          next_phase := 9000;
        ELSE
          (* Recalculate schedule with shifted base time *)
          next_phase := 1010;
        END_IF;
      ELSE
        (* Stage 0 fits → proceed to stage 1+ tasks *)
        IF w_task_cnt = 0 THEN
          next_phase := 8000;  (* No more tasks → ACTIVATE *)
        ELSE
          cur_task_idx := 1;
          next_phase := 2001;
        END_IF;
      END_IF;
    ELSE
      (* Stage 0 doesn't fit → REJECT this batch *)
      next_phase := 9000;
    END_IF;
  END_IF;

(* ════════════════════════════════════════════════════════════ *)
(* PHASE 2001: FIT_TASK — fit stage 1+ tasks one per tick      *)
(* ════════════════════════════════════════════════════════════ *)
ELSIF phase = 2001 THEN
  IF cur_task_idx > w_task_cnt THEN
    (* All tasks fit → ACTIVATE *)
    next_phase := 8000;
  ELSE
    (* Get current task data *)
    si := w_tasks[cur_task_idx].stage;
    ti := w_trans[cur_task_idx];

    (* Overlap delay check *)
    fb_ovlp_delay(
      i_lift_stn   := w_tasks[cur_task_idx].lift_station,
      i_sink_stn   := w_tasks[cur_task_idx].sink_station,
      i_trans_id   := ti,
      i_task_start := w_tasks[cur_task_idx].start_time,
      i_task_end   := w_tasks[cur_task_idx].finish_time,
      i_margin_s   := CONFLICT_MARGIN_S
    );
    ovlp_delay_s := fb_ovlp_delay.o_delay_s;

    (* Idle-slot fit check *)
    fb_fit(
      i_lift_stn     := w_tasks[cur_task_idx].lift_station,
      i_sink_stn     := w_tasks[cur_task_idx].sink_station,
      i_trans_id     := ti,
      i_task_start   := w_tasks[cur_task_idx].start_time,
      i_task_end     := w_tasks[cur_task_idx].finish_time,
      i_shift_s      := ovlp_delay_s,
      i_calc_time_s  := w_tasks[cur_task_idx].calc_time,
      i_max_time_s   := w_tasks[cur_task_idx].max_time,
      i_flex_factor  := FLEX_FACTOR,
      i_margin_s     := MARGIN_S
    );

    total_delay_s := ovlp_delay_s + fb_fit.o_result.delay_s;

    IF fb_fit.o_result.fits THEN
      IF total_delay_s <= MARGIN_S THEN
        (* Fits with negligible delay → next task *)
        cur_task_idx := cur_task_idx + 1;
        next_phase := 2001;
      ELSE
        (* Delay needed → record and recalculate *)
        delay_stage  := si;
        delay_amount := total_delay_s;
        delay_target := 1;   (* program stage *)
        next_phase   := 3000;
      END_IF;
    ELSE
      (* Does not fit → REJECT (simplified: no backward chaining) *)
      next_phase := 9000;
    END_IF;
  END_IF;

(* ════════════════════════════════════════════════════════════ *)
(* PHASE 3000: APPLY_DELAY — write delay to program, recalc   *)
(* ════════════════════════════════════════════════════════════ *)
ELSIF phase = 3000 THEN
  fit_round := fit_round + 1;
  IF fit_round > MAX_FIT_ROUNDS THEN
    next_phase := 9000;
  ELSE
    IF delay_target = 0 THEN
      (* Stage 0 delay: shift base time (handled in FIT_STAGE0, shouldn't reach here) *)
      sched_base_time := sched_base_time + delay_amount;
    ELSIF delay_target = 1 THEN
      (* Program stage delay: increase cal_time *)
      prog_idx := delay_stage;
      IF prog_idx >= 1 AND prog_idx <= 30 THEN
        old_cal := g_programs[cur_wait_unit].stages[prog_idx].cal_time;
        max_cal := g_programs[cur_wait_unit].stages[prog_idx].max_time;
        new_cal := old_cal + REAL_TO_INT(delay_amount);
        IF new_cal > max_cal AND max_cal > 0 THEN
          new_cal := max_cal;
        END_IF;
        g_programs[cur_wait_unit].stages[prog_idx].cal_time := new_cal;
      END_IF;
    END_IF;
    (* Recalculate: schedule → tasks → idle → fit *)
    next_phase := 1010;
  END_IF;

(* ════════════════════════════════════════════════════════════ *)
(* PHASE 8000: ACTIVATE — commit changes to pending write      *)
(* ════════════════════════════════════════════════════════════ *)
ELSIF phase = 8000 THEN
  (* Store pending write data *)
  FOR ui := 1 TO 10 DO
    g_dep_pending.programs[ui] := g_programs[ui];
    g_dep_pending.schedule[ui] := g_schedule[ui];
  END_FOR;
  g_dep_pending.batch_unit  := cur_wait_unit;
  g_dep_pending.batch_stage := 0;    (* 90 → 0 *)
  g_dep_pending.time_s      := i_time_s;
  g_dep_pending.valid        := TRUE;

  (* Restore globals from sandbox (undo DEP's temp changes) *)
  fb_sandbox(i_cmd := 2);
  fb_sandbox(i_cmd := 3);   (* clear sandbox *)

  g_dep_activated := TRUE;
  o_activated := TRUE;

  next_phase := 8010;

(* ════════════════════════════════════════════════════════════ *)
(* PHASE 8010: WAIT_SAVE — wait for TSK to process pending     *)
(* ════════════════════════════════════════════════════════════ *)
ELSIF phase = 8010 THEN
  IF NOT g_dep_pending.valid THEN
    (* TSK has processed the pending write *)
    next_phase := 8020;
  END_IF;
  (* Otherwise keep waiting *)

(* ════════════════════════════════════════════════════════════ *)
(* PHASE 8020: END_DELAY — stabilization ticks                 *)
(* ════════════════════════════════════════════════════════════ *)
ELSIF phase = 8020 THEN
  end_delay_cnt := 0;
  next_phase := 8021;

ELSIF phase >= 8021 AND phase <= 8120 THEN
  end_delay_cnt := end_delay_cnt + 1;
  IF end_delay_cnt >= END_DELAY_TICKS THEN
    next_phase := 8100;
  ELSE
    next_phase := phase + 1;
    IF next_phase > 8120 THEN
      next_phase := 8100;
    END_IF;
  END_IF;

(* ════════════════════════════════════════════════════════════ *)
(* PHASE 8100: RESTART — back to WAIT_STABLE                   *)
(* ════════════════════════════════════════════════════════════ *)
ELSIF phase = 8100 THEN
  g_dep_activated := FALSE;
  next_phase := 1;

(* ════════════════════════════════════════════════════════════ *)
(* PHASE 9000: REJECT — restore, try next batch                *)
(* ════════════════════════════════════════════════════════════ *)
ELSIF phase = 9000 THEN
  (* Restore globals from sandbox (undo changes for this batch) *)
  fb_sandbox(i_cmd := 2);

  (* Try next waiting batch *)
  cur_wait_idx := cur_wait_idx + 1;
  IF cur_wait_idx > waiting_cnt THEN
    (* No more batches → back to waiting *)
    fb_sandbox(i_cmd := 3);
    next_phase := 1;
  ELSE
    (* Try next batch — re-snapshot is still valid *)
    next_phase := 1000;
  END_IF;

(* ════════════════════════════════════════════════════════════ *)
(* Unknown phase → reset                                       *)
(* ════════════════════════════════════════════════════════════ *)
ELSE
  next_phase := 1;
END_IF;

(* ── Phase assignment ── *)
phase := next_phase;
o_phase := phase;
          
END_FUNCTION_BLOCK

FUNCTION_BLOCK SIM_FB_XMotion
  VAR_INPUT
    delta_t : REAL;
    x_target : REAL;
    x_min : REAL;
    x_max : REAL;
    v_max : REAL;
    t_acc : REAL;
    t_dec : REAL;
  END_VAR
  VAR_OUTPUT
    arrived : BOOL;
  END_VAR
  VAR_IN_OUT
    x_pos : REAL;
    v_x : REAL;
  END_VAR
  VAR
    drive_target : REAL;
    distance : REAL;
    dir : REAL;
    a_acc : REAL;
    a_dec : REAL;
    brake_dist : REAL;
    new_vel : REAL;
    travel : REAL;
  END_VAR

            IF (x_max > x_min) THEN
  IF x_pos < x_min THEN
    drive_target := x_min;
  ELSIF x_pos > x_max THEN
    drive_target := x_max;
  ELSE
    IF x_target < x_min THEN
      drive_target := x_min;
    ELSIF x_target > x_max THEN
      drive_target := x_max;
    ELSE
      drive_target := x_target;
    END_IF;
  END_IF;
ELSE
  drive_target := x_target;
END_IF;

arrived := ABS(x_pos - drive_target) <= 3.0;
IF arrived THEN
  x_pos := drive_target;
  v_x := 0.0;
  RETURN;
END_IF;

IF t_acc <= 0.0 THEN t_acc := 0.001; END_IF;
IF t_dec <= 0.0 THEN t_dec := 0.001; END_IF;
IF v_max < 0.0 THEN v_max := 0.0; END_IF;

a_acc := v_max / t_acc;
a_dec := v_max / t_dec;

dir := 1.0;
IF drive_target < x_pos THEN
  dir := -1.0;
END_IF;

distance := ABS(drive_target - x_pos);

IF a_dec > 0.0 THEN
  brake_dist := (v_x * v_x) / (2.0 * a_dec);
ELSE
  brake_dist := 0.0;
END_IF;

IF brake_dist >= distance THEN
  new_vel := v_x - a_dec * delta_t;
  IF new_vel < 0.0 THEN new_vel := 0.0; END_IF;
ELSE
  new_vel := v_x + a_acc * delta_t;
  IF new_vel > v_max THEN new_vel := v_max; END_IF;
END_IF;

travel := new_vel * delta_t;
IF travel >= distance THEN
  x_pos := drive_target;
  v_x := 0.0;
  arrived := TRUE;
ELSE
  x_pos := x_pos + dir * travel;
  v_x := new_vel;
  arrived := FALSE;
END_IF;
          
END_FUNCTION_BLOCK

FUNCTION_BLOCK SIM_FB_ZMotion
  VAR_INPUT
    delta_t : REAL;
    station_type : INT;
    z_total_mm : REAL;
    z_slow_dry_mm : REAL;
    z_slow_wet_mm : REAL;
    z_slow_end_mm : REAL;
    z_slow_mm_s : REAL;
    z_fast_mm_s : REAL;
    drip_delay_s : REAL;
  END_VAR
  VAR_OUTPUT
    done : BOOL;
  END_VAR
  VAR_IN_OUT
    z_mm : REAL;
    z_stage : INT;
    z_timer_s : REAL;
  END_VAR
  VAR_EXTERNAL
    STN_WET : INT;
  END_VAR
  VAR
    slow_zone : REAL;
  END_VAR

            done := FALSE;

(* Select slow zone based on station type *)
IF station_type = STN_WET THEN
  slow_zone := z_slow_wet_mm;
ELSE
  slow_zone := z_slow_dry_mm;
END_IF;

CASE z_stage OF

  (* === LIFT: stages 1-5 — nosto altaasta ylös === *)

  1: (* Init delay: device_delay + dropping_time *)
    z_timer_s := z_timer_s - delta_t;
    IF z_timer_s <= 0.0 THEN
      z_stage := 2;
      z_mm := z_total_mm;
    END_IF;

  2: (* Slow lift start — hidas nosto nesteestä *)
    z_mm := z_mm - z_slow_mm_s * delta_t;
    IF z_mm <= (z_total_mm - slow_zone) THEN
      z_stage := 3;
    END_IF;

  3: (* Fast lift — nopea nosto *)
    z_mm := z_mm - z_fast_mm_s * delta_t;
    IF z_mm <= z_slow_end_mm THEN
      z_stage := 4;
    END_IF;

  4: (* Slow lift end — hidas loppunosto *)
    z_mm := z_mm - z_slow_mm_s * delta_t;
    IF z_mm <= 0.0 THEN
      z_mm := 0.0;
      z_timer_s := drip_delay_s;
      z_stage := 5;
    END_IF;

  5: (* Drip delay — tippumisviive yläasemassa *)
    z_timer_s := z_timer_s - delta_t;
    IF z_timer_s <= 0.0 THEN
      z_stage := 0;
      done := TRUE;
    END_IF;

  (* === SINK: stages 6-8 — lasku altaaseen === *)

  6: (* Init delay: device_delay + drip_delay *)
    z_timer_s := z_timer_s - delta_t;
    IF z_timer_s <= 0.0 THEN
      z_stage := 7;
    END_IF;

  7: (* Fast sink — nopea lasku *)
    z_mm := z_mm + z_fast_mm_s * delta_t;
    IF z_mm >= (z_total_mm - slow_zone) THEN
      z_stage := 8;
    END_IF;

  8: (* Slow sink — hidas lasku nesteeseen *)
    z_mm := z_mm + z_slow_mm_s * delta_t;
    IF z_mm >= z_total_mm THEN
      z_mm := z_total_mm;
      z_stage := 0;
      done := TRUE;
    END_IF;

END_CASE;
          
END_FUNCTION_BLOCK

FUNCTION_BLOCK STC_FB_FindStation
  VAR_INPUT
    station_number : INT;
  END_VAR
  VAR_OUTPUT
    found : BOOL;
    idx : INT;
    x_mm : REAL;
    stype : INT;
    device_delay_s : REAL;
    dropping_time_s : REAL;
  END_VAR
  VAR_EXTERNAL
    g_stations : ARRAY[101..125] OF STATION_T;
  END_VAR
  VAR
    st : STATION_T;
  END_VAR

            (* Direct lookup by station number — no loop needed *)
IF (station_number >= 101) AND (station_number <= 125) THEN
  st := g_stations[station_number];
  IF st.tank_id <> 0 THEN
    found := TRUE;
    idx := station_number;
    x_mm := st.x_position;
    stype := st.stn_type;
    device_delay_s := st.device_delay;
    dropping_time_s := st.dropping_time;
    RETURN;
  END_IF;
END_IF;

found := FALSE;
idx := 0;
x_mm := 0.0;
stype := 0;
device_delay_s := 0.0;
dropping_time_s := 0.0;
          
END_FUNCTION_BLOCK

FUNCTION_BLOCK STC_FB_MeasureMoveTimes
  VAR_INPUT
    t_id : INT;
    phase : INT;
    delta_t : REAL;
    vel_x : REAL;
    z_stage : INT;
    lift_stn : INT;
    sink_stn : INT;
    from_stn : INT;
  END_VAR
  VAR_EXTERNAL
    g_move : ARRAY[1..3] OF MOVE_TIMES_T;
  END_VAR
  VAR
    prev_phase : INT := -1;
    timer : REAL := 0.0;
    travel_from : INT;
    travel_to : INT;
    lift_idx : INT;
    sink_idx : INT;
  END_VAR

            (* ---- Phase transition detection ---- *)
IF phase <> prev_phase THEN

  (* -- Save completed measurement and set up next -- *)

  IF prev_phase = 1 AND phase = 2 THEN
    (* Travel to lift complete → save travel time *)
    IF travel_from >= 1 AND travel_from <= 25
       AND travel_to >= 1 AND travel_to <= 25 THEN
      g_move[t_id].travel[travel_from].to_s[travel_to] := timer;
    END_IF;
    (* Start timing lift — timer starts at 0, accumulates only in z_stage 2-4 *)
    lift_idx := lift_stn - 100;
    timer := 0.0;

  ELSIF prev_phase = 2 AND phase = 3 THEN
    (* Lift complete → save lift time (pure mechanical Z-motion only) *)
    IF lift_idx >= 1 AND lift_idx <= 25 THEN
      g_move[t_id].lift_s[lift_idx] := timer;
    END_IF;
    (* Start timing travel to sink *)
    travel_from := lift_stn - 100;
    travel_to := sink_stn - 100;
    timer := 0.0;

  ELSIF prev_phase = 3 AND phase = 4 THEN
    (* Travel to sink complete → save travel time *)
    IF travel_from >= 1 AND travel_from <= 25
       AND travel_to >= 1 AND travel_to <= 25 THEN
      g_move[t_id].travel[travel_from].to_s[travel_to] := timer;
    END_IF;
    (* Start timing sink — timer starts at 0, accumulates only in z_stage 7-8 *)
    sink_idx := sink_stn - 100;
    timer := 0.0;

  ELSIF prev_phase = 4 AND phase = 0 THEN
    (* Sink complete → save sink time (pure mechanical Z-motion only) *)
    IF sink_idx >= 1 AND sink_idx <= 25 THEN
      g_move[t_id].sink_s[sink_idx] := timer;
    END_IF;
    timer := 0.0;

  ELSIF prev_phase = 0 AND phase = 1 THEN
    (* New cycle starting → set up travel-to-lift *)
    travel_from := from_stn - 100;
    travel_to := lift_stn - 100;
    timer := 0.0;

  ELSE
    (* Unexpected transition → just reset *)
    timer := 0.0;
  END_IF;

  prev_phase := phase;

ELSE
  (* ---- No transition: accumulate timer ---- *)

  IF phase = 1 OR phase = 3 THEN
    (* Travel: only count time when actually moving *)
    (* Filters out TWA collision avoidance stops    *)
    IF ABS(vel_x) > 0.1 THEN
      timer := timer + delta_t;
    END_IF;

  ELSIF phase = 2 THEN
    (* Lift: only mechanical Z-motion stages 2-4 *)
    (* Excludes: stage 1 (device_delay + dropping_time), stage 5 (drip_delay) *)
    IF z_stage >= 2 AND z_stage <= 4 THEN
      timer := timer + delta_t;
    END_IF;

  ELSIF phase = 4 THEN
    (* Sink: only mechanical Z-motion stages 7-8 *)
    (* Excludes: stage 6 (device_delay + drip_delay) *)
    IF z_stage >= 7 AND z_stage <= 8 THEN
      timer := timer + delta_t;
    END_IF;
  END_IF;

END_IF;
          
END_FUNCTION_BLOCK

FUNCTION_BLOCK TSK_FB_Analyze
  VAR_OUTPUT
    o_has_conflict : BOOL;
    o_conf_type : INT;
    o_conf_unit : INT;
    o_conf_stage : INT;
    o_conf_trans : INT;
    o_blocked_unit : INT;
    o_blocked_stage : INT;
    o_deficit : REAL;
    checked_count : INT;
  END_VAR
  VAR_EXTERNAL
    g_tasks : ARRAY[1..3] OF TSK_QUEUE_T;
    g_stations : ARRAY[101..125] OF STATION_T;
  END_VAR
  VAR
    sorted : ARRAY[1..30] OF TSK_TASK_T;
    sorted_trans : ARRAY[1..30] OF INT;
    sorted_cnt : INT;
    chk : ARRAY[1..30] OF TSK_CHECKED_T;
    chk_cnt : INT;
    ti : INT;
    qi : INT;
    si : INT;
    ins : INT;
    ci : INT;
    tmp_task : TSK_TASK_T;
    tmp_tid : INT;
    prev_sink : INT;
    next_lift : INT;
    travel_s : REAL;
    gap_s : REAL;
    deficit_s : REAL;
    calc_t : REAL;
    min_t : REAL;
    max_t : REAL;
    f_down : REAL;
    f_up : REAL;
    x1_min : REAL;
    x1_max : REAL;
    x2_min : REAL;
    x2_max : REAL;
    xo_start : REAL;
    xo_end : REAL;
    to_start : REAL;
    to_end : REAL;
    lift_x : REAL;
    sink_x : REAL;
    l_idx : INT;
    s_idx : INT;
    DEFICIT_TOL : REAL := 1.0;
    fb_travel : STC_FB_CalcHorizontalTravel;
  END_VAR

            o_has_conflict := FALSE;
o_conf_type    := 0;
o_deficit      := 0.0;
checked_count  := 0;
chk_cnt        := 0;

(* ══════ Step 1: Merge all queues into sorted[] by start_time (insertion sort) ══════ *)
sorted_cnt := 0;
FOR ti := 1 TO 3 DO
  FOR qi := 1 TO g_tasks[ti].count DO
    IF g_tasks[ti].queue[qi].unit > 0 THEN
      (* Insert into sorted position *)
      sorted_cnt := sorted_cnt + 1;
      IF sorted_cnt <= 30 THEN
        sorted[sorted_cnt] := g_tasks[ti].queue[qi];
        sorted_trans[sorted_cnt] := ti;
        (* Insertion sort: bubble up *)
        ins := sorted_cnt;
        WHILE ins > 1 DO
          IF sorted[ins].start_time < sorted[ins - 1].start_time THEN
            tmp_task := sorted[ins];
            tmp_tid  := sorted_trans[ins];
            sorted[ins] := sorted[ins - 1];
            sorted_trans[ins] := sorted_trans[ins - 1];
            sorted[ins - 1] := tmp_task;
            sorted_trans[ins - 1] := tmp_tid;
            ins := ins - 1;
          ELSE
            ins := 0; (* break *)
          END_IF;
        END_WHILE;
      END_IF;
    END_IF;
  END_FOR;
END_FOR;

IF sorted_cnt = 0 THEN RETURN; END_IF;

(* ══════ Step 2: Walk sorted list, build checked[], detect conflicts ══════ *)
FOR si := 1 TO sorted_cnt DO

  (* Calculate flex for this task *)
  calc_t := sorted[si].calc_time;
  min_t  := sorted[si].min_time;
  max_t  := sorted[si].max_time;
  f_down := calc_t - min_t;
  IF f_down < 0.0 THEN f_down := 0.0; END_IF;
  f_up := max_t - calc_t;
  IF f_up < 0.0 THEN f_up := 0.0; END_IF;

  (* Get X range for this task *)
  l_idx := sorted[si].lift_station - 100;
  s_idx := sorted[si].sink_station - 100;
  IF l_idx >= 1 AND l_idx <= 25 THEN
    lift_x := g_stations[sorted[si].lift_station].x_position;
  ELSE
    lift_x := 0.0;
  END_IF;
  IF s_idx >= 1 AND s_idx <= 25 THEN
    sink_x := g_stations[sorted[si].sink_station].x_position;
  ELSE
    sink_x := 0.0;
  END_IF;
  IF lift_x < sink_x THEN
    x1_min := lift_x;
    x1_max := sink_x;
  ELSE
    x1_min := sink_x;
    x1_max := lift_x;
  END_IF;

  (* Add to checked list *)
  chk_cnt := chk_cnt + 1;
  IF chk_cnt <= 30 THEN
    chk[chk_cnt].unit        := sorted[si].unit;
    chk[chk_cnt].stage       := sorted[si].stage;
    chk[chk_cnt].transporter := sorted_trans[si];
    chk[chk_cnt].start_time  := sorted[si].start_time;
    chk[chk_cnt].end_time    := sorted[si].finish_time;
    chk[chk_cnt].flex_down   := f_down;
    chk[chk_cnt].flex_up     := f_up;
    chk[chk_cnt].x_min       := x1_min;
    chk[chk_cnt].x_max       := x1_max;
    chk[chk_cnt].is_conflict := FALSE;
  END_IF;

  (* ─── Check TASK_SEQUENCE: same transporter, previous task ─── *)
  (* Find the previous task for this transporter in sorted order *)
  FOR ci := si - 1 TO 1 BY -1 DO
    IF sorted_trans[ci] = sorted_trans[si] THEN
      (* Found previous task on same transporter *)
      prev_sink := sorted[ci].sink_station;
      next_lift := sorted[si].lift_station;

      fb_travel(i_from_stn := prev_sink, i_to_stn := next_lift, i_trans := sorted_trans[si]);
      travel_s := fb_travel.o_travel_s;

      gap_s := sorted[si].start_time - sorted[ci].finish_time;
      deficit_s := travel_s - gap_s;

      IF deficit_s > DEFICIT_TOL THEN
        (* TASK_SEQUENCE conflict! *)
        o_has_conflict  := TRUE;
        o_conf_type     := 1;
        o_conf_unit     := sorted[si].unit;
        o_conf_stage    := sorted[si].stage;
        o_conf_trans    := sorted_trans[si];
        o_blocked_unit  := sorted[ci].unit;
        o_blocked_stage := sorted[ci].stage;
        o_deficit       := deficit_s;
        IF chk_cnt <= 30 THEN
          chk[chk_cnt].is_conflict := TRUE;
        END_IF;
        checked_count := chk_cnt;
        RETURN;
      END_IF;

      EXIT; (* only check immediate predecessor *)
    END_IF;
  END_FOR;

  (* ─── Check TRANSPORTER_COLLISION: different transporter, X+time overlap ─── *)
  FOR ci := 1 TO chk_cnt - 1 DO
    IF chk[ci].transporter <> sorted_trans[si] THEN
      (* X overlap *)
      x2_min := chk[ci].x_min;
      x2_max := chk[ci].x_max;
      xo_start := x1_min;
      IF x2_min > xo_start THEN xo_start := x2_min; END_IF;
      xo_end := x1_max;
      IF x2_max < xo_end THEN xo_end := x2_max; END_IF;

      IF xo_start < xo_end THEN
        (* Time overlap *)
        to_start := sorted[si].start_time;
        IF chk[ci].start_time > to_start THEN to_start := chk[ci].start_time; END_IF;
        to_end := sorted[si].finish_time;
        IF chk[ci].end_time < to_end THEN to_end := chk[ci].end_time; END_IF;

        IF to_start < to_end THEN
          (* TRANSPORTER_COLLISION conflict! *)
          deficit_s := (to_end - to_start) + 2.0; (* +2s margin *)
          o_has_conflict  := TRUE;
          o_conf_type     := 2;
          o_conf_unit     := sorted[si].unit;
          o_conf_stage    := sorted[si].stage;
          o_conf_trans    := sorted_trans[si];
          o_blocked_unit  := chk[ci].unit;
          o_blocked_stage := chk[ci].stage;
          o_deficit       := deficit_s;
          IF chk_cnt <= 30 THEN
            chk[chk_cnt].is_conflict := TRUE;
          END_IF;
          checked_count := chk_cnt;
          RETURN;
        END_IF;
      END_IF;
    END_IF;
  END_FOR;

END_FOR;

(* No conflict found *)
checked_count := chk_cnt;
          
END_FUNCTION_BLOCK

FUNCTION_BLOCK TSK_FB_NoTreatment
  VAR_INPUT
    i_time_s : REAL;
  END_VAR
  VAR_EXTERNAL
    g_units : ARRAY[1..10] OF UNIT_T;
    g_state : ARRAY[1..3] OF TRANSPORTER_STATE_T;
    g_cfg : ARRAY[1..3] OF TRANSPORTER_CFG_T;
    g_tasks : ARRAY[1..3] OF TSK_QUEUE_T;
    g_stations : ARRAY[101..125] OF STATION_T;
    g_station_count : INT;
  END_VAR
  VAR
    ui : INT;
    ai : INT;
    qi : INT;
    loc : INT;
    tgt : INT;
    cov_t : INT;
    area : TASK_AREA_T;
    dest_stn : INT;
    si : INT;
    stn_free : BOOL;
    stn_ok : BOOL;
    xfer_s : REAL;
    task_start : REAL;
    task_end : REAL;
    fb_find : STC_FB_FindTransporter;
    fb_xfer : STC_FB_CalcTransferTime;
  END_VAR

            FOR ui := 1 TO 10 DO
  tgt := g_units[ui].target;
  loc := g_units[ui].location;

  (* Skip: no target, target is process (handled by schedule), not on station *)
  IF tgt <> 0 AND tgt <> 3 AND loc >= 100 THEN
    (* Find covering transporter *)
    fb_find(i_lift_stn := loc, i_sink_stn := 0);
    cov_t := fb_find.o_trans_id;

    IF cov_t >= 1 AND cov_t <= 3 THEN
      (* Check transporter is idle: phase=0, active *)
      IF g_state[cov_t].phase = 0 AND g_state[cov_t].active THEN

        (* Find destination station: first available in transporter area *)
        dest_stn := 0;
        FOR ai := 1 TO 4 DO
          IF dest_stn = 0 THEN
            area := g_cfg[cov_t].task_area[ai];
            IF area.min_sink > 0 THEN
              FOR si := area.min_sink TO area.max_sink DO
                IF dest_stn = 0 AND si <> loc AND si >= 101 AND si <= 125 THEN
                  (* Check station is free: no unit there *)
                  stn_free := TRUE;
                  FOR qi := 1 TO 10 DO
                    IF g_units[qi].location = si AND g_units[qi].status = 1 THEN
                      stn_free := FALSE;
                    END_IF;
                  END_FOR;
                  IF stn_free THEN
                    dest_stn := si;
                  END_IF;
                END_IF;
              END_FOR;
            END_IF;
          END_IF;
        END_FOR;

        IF dest_stn > 0 THEN
          (* Calculate timing *)
          fb_xfer(i_from_stn := loc, i_to_stn := dest_stn, i_trans := cov_t);
          xfer_s := fb_xfer.o_total_s;

          task_start := i_time_s;
          task_end   := task_start + xfer_s;

          (* Append to queue *)
          qi := g_tasks[cov_t].count + 1;
          IF qi <= 10 THEN
            g_tasks[cov_t].queue[qi].unit         := ui;
            g_tasks[cov_t].queue[qi].stage        := 0;  (* no program stage *)
            g_tasks[cov_t].queue[qi].lift_station := loc;
            g_tasks[cov_t].queue[qi].sink_station := dest_stn;
            g_tasks[cov_t].queue[qi].start_time   := task_start;
            g_tasks[cov_t].queue[qi].finish_time  := task_end;
            g_tasks[cov_t].queue[qi].calc_time    := 0.0;
            g_tasks[cov_t].queue[qi].min_time     := 0.0;
            g_tasks[cov_t].queue[qi].max_time     := 0.0;
            g_tasks[cov_t].count := qi;
          END_IF;
        END_IF;

      END_IF; (* transporter idle *)
    END_IF; (* covering transporter found *)
  END_IF; (* valid target *)
END_FOR;
          
END_FUNCTION_BLOCK

FUNCTION_BLOCK TSK_FB_Resolve
  VAR_INPUT
    i_conf_unit : INT;
    i_conf_stage : INT;
    i_conf_trans : INT;
    i_blocked_unit : INT;
    i_blocked_stage : INT;
    i_deficit : REAL;
  END_VAR
  VAR_OUTPUT
    o_solved : BOOL;
    o_total_delay : REAL;
    o_total_adv : REAL;
  END_VAR
  VAR_EXTERNAL
    g_tasks : ARRAY[1..3] OF TSK_QUEUE_T;
    g_schedule : ARRAY[1..10] OF TSK_SCHEDULE_T;
    g_batches : ARRAY[1..10] OF BATCH_T;
  END_VAR
  VAR
    remain : REAL;
    cap : REAL;
    flex : REAL;
    amount : REAL;
    qi : INT;
    si : INT;
    cnt : INT;
    sc : INT;
    locks : ARRAY[1..50] OF INT;
    lock_dir : ARRAY[1..50] OF INT;
    lock_cnt : INT;
    lock_key : INT;
    is_locked : BOOL;
    lock_i : INT;
    prev_flex : REAL;
    next_flex : REAL;
    prev_stage_flex : REAL;
  END_VAR

            o_solved      := FALSE;
o_total_delay := 0.0;
o_total_adv   := 0.0;
remain        := i_deficit;

IF remain <= 0.1 THEN
  o_solved := TRUE;
  RETURN;
END_IF;

(* ══════ Phase 1: ADVANCE prev batch (blocked_unit, blocked_stage) ══════ *)
(* Reduce treatment time toward min_time = flex_down *)

(* Find flex_down for blocked stage in schedule *)
prev_flex := 0.0;
IF i_blocked_unit >= 1 AND i_blocked_unit <= 10 THEN
  sc := g_schedule[i_blocked_unit].stage_count;
  FOR si := 1 TO sc DO
    IF si = i_blocked_stage THEN
      prev_flex := g_schedule[i_blocked_unit].stages[si].calc_time
                 - g_schedule[i_blocked_unit].stages[si].min_time;
      IF prev_flex < 0.0 THEN prev_flex := 0.0; END_IF;
    END_IF;
  END_FOR;
END_IF;

IF prev_flex > 0.1 THEN
  (* Cap: 90% if batch is on this stage, 50% otherwise *)
  IF g_batches[i_blocked_unit].cur_stage = i_blocked_stage THEN
    cap := 0.9;
  ELSE
    cap := 0.5;
  END_IF;
  amount := prev_flex * cap;
  IF amount > remain THEN amount := remain; END_IF;

  (* Apply: shift blocked batch's stage exit earlier *)
  IF i_blocked_stage >= 1 AND i_blocked_stage <= 30 THEN
    g_schedule[i_blocked_unit].stages[i_blocked_stage].calc_time :=
      g_schedule[i_blocked_unit].stages[i_blocked_stage].calc_time - amount;
    g_schedule[i_blocked_unit].stages[i_blocked_stage].exit_time :=
      g_schedule[i_blocked_unit].stages[i_blocked_stage].exit_time - amount;
    (* Propagate: shift all later stages earlier *)
    sc := g_schedule[i_blocked_unit].stage_count;
    FOR si := i_blocked_stage + 1 TO sc DO
      g_schedule[i_blocked_unit].stages[si].entry_time :=
        g_schedule[i_blocked_unit].stages[si].entry_time - amount;
      g_schedule[i_blocked_unit].stages[si].exit_time :=
        g_schedule[i_blocked_unit].stages[si].exit_time - amount;
    END_FOR;
  END_IF;

  (* Update tasks for blocked unit in all transporter queues *)
  FOR qi := 1 TO 3 DO
    FOR si := 1 TO g_tasks[qi].count DO
      IF g_tasks[qi].queue[si].unit = i_blocked_unit
         AND g_tasks[qi].queue[si].stage >= i_blocked_stage THEN
        g_tasks[qi].queue[si].start_time :=
          g_tasks[qi].queue[si].start_time - amount;
        g_tasks[qi].queue[si].finish_time :=
          g_tasks[qi].queue[si].finish_time - amount;
      END_IF;
    END_FOR;
  END_FOR;

  remain := remain - amount;
  o_total_adv := o_total_adv + amount;
END_IF;

IF remain <= 0.1 THEN
  o_solved := TRUE;
  RETURN;
END_IF;

(* ══════ Phase 2: DELAY next batch conflict stage (conf_unit, conf_stage) ══════ *)
(* Increase treatment time toward max_time = flex_up *)
next_flex := 0.0;
IF i_conf_unit >= 1 AND i_conf_unit <= 10 AND i_conf_stage >= 1 AND i_conf_stage <= 30 THEN
  next_flex := g_schedule[i_conf_unit].stages[i_conf_stage].max_time
             - g_schedule[i_conf_unit].stages[i_conf_stage].calc_time;
  IF next_flex < 0.0 THEN next_flex := 0.0; END_IF;
END_IF;

IF next_flex > 0.1 THEN
  IF g_batches[i_conf_unit].cur_stage = i_conf_stage THEN
    cap := 0.9;
  ELSE
    cap := 0.5;
  END_IF;
  amount := next_flex * cap;
  IF amount > remain THEN amount := remain; END_IF;

  (* Apply: extend conflict stage, shift later stages forward *)
  g_schedule[i_conf_unit].stages[i_conf_stage].calc_time :=
    g_schedule[i_conf_unit].stages[i_conf_stage].calc_time + amount;
  g_schedule[i_conf_unit].stages[i_conf_stage].exit_time :=
    g_schedule[i_conf_unit].stages[i_conf_stage].exit_time + amount;
  sc := g_schedule[i_conf_unit].stage_count;
  FOR si := i_conf_stage + 1 TO sc DO
    g_schedule[i_conf_unit].stages[si].entry_time :=
      g_schedule[i_conf_unit].stages[si].entry_time + amount;
    g_schedule[i_conf_unit].stages[si].exit_time :=
      g_schedule[i_conf_unit].stages[si].exit_time + amount;
  END_FOR;

  (* Update tasks *)
  FOR qi := 1 TO 3 DO
    FOR si := 1 TO g_tasks[qi].count DO
      IF g_tasks[qi].queue[si].unit = i_conf_unit
         AND g_tasks[qi].queue[si].stage >= i_conf_stage THEN
        g_tasks[qi].queue[si].start_time :=
          g_tasks[qi].queue[si].start_time + amount;
        g_tasks[qi].queue[si].finish_time :=
          g_tasks[qi].queue[si].finish_time + amount;
      END_IF;
    END_FOR;
  END_FOR;

  remain := remain - amount;
  o_total_delay := o_total_delay + amount;
END_IF;

IF remain <= 0.1 THEN
  o_solved := TRUE;
  RETURN;
END_IF;

(* ══════ Phase 3: DELAY next batch previous stage (conf_stage - 1) ══════ *)
IF i_conf_stage > 1 THEN
  prev_stage_flex := 0.0;
  IF i_conf_unit >= 1 AND i_conf_unit <= 10 AND (i_conf_stage - 1) >= 1 THEN
    prev_stage_flex := g_schedule[i_conf_unit].stages[i_conf_stage - 1].max_time
                     - g_schedule[i_conf_unit].stages[i_conf_stage - 1].calc_time;
    IF prev_stage_flex < 0.0 THEN prev_stage_flex := 0.0; END_IF;
  END_IF;

  IF prev_stage_flex > 0.1 THEN
    IF g_batches[i_conf_unit].cur_stage = (i_conf_stage - 1) THEN
      cap := 0.9;
    ELSE
      cap := 0.5;
    END_IF;
    amount := prev_stage_flex * cap;
    IF amount > remain THEN amount := remain; END_IF;

    (* Apply: extend previous stage, propagate from conf_stage onward *)
    g_schedule[i_conf_unit].stages[i_conf_stage - 1].calc_time :=
      g_schedule[i_conf_unit].stages[i_conf_stage - 1].calc_time + amount;
    g_schedule[i_conf_unit].stages[i_conf_stage - 1].exit_time :=
      g_schedule[i_conf_unit].stages[i_conf_stage - 1].exit_time + amount;
    sc := g_schedule[i_conf_unit].stage_count;
    FOR si := i_conf_stage TO sc DO
      g_schedule[i_conf_unit].stages[si].entry_time :=
        g_schedule[i_conf_unit].stages[si].entry_time + amount;
      g_schedule[i_conf_unit].stages[si].exit_time :=
        g_schedule[i_conf_unit].stages[si].exit_time + amount;
    END_FOR;

    FOR qi := 1 TO 3 DO
      FOR si := 1 TO g_tasks[qi].count DO
        IF g_tasks[qi].queue[si].unit = i_conf_unit
           AND g_tasks[qi].queue[si].stage >= (i_conf_stage - 1) THEN
          g_tasks[qi].queue[si].start_time :=
            g_tasks[qi].queue[si].start_time + amount;
          g_tasks[qi].queue[si].finish_time :=
            g_tasks[qi].queue[si].finish_time + amount;
        END_IF;
      END_FOR;
    END_FOR;

    remain := remain - amount;
    o_total_delay := o_total_delay + amount;
  END_IF;
END_IF;

IF remain <= 0.1 THEN
  o_solved := TRUE;
  RETURN;
END_IF;

(* ══════ Phase 4: DELAY prev past next (forced reorder) ══════ *)
(* Delay blocked_unit's stage to push it past conflict *)
prev_flex := 0.0;
IF i_blocked_unit >= 1 AND i_blocked_unit <= 10 AND i_blocked_stage >= 1 AND i_blocked_stage <= 30 THEN
  prev_flex := g_schedule[i_blocked_unit].stages[i_blocked_stage].max_time
             - g_schedule[i_blocked_unit].stages[i_blocked_stage].calc_time;
  IF prev_flex < 0.0 THEN prev_flex := 0.0; END_IF;
END_IF;

IF prev_flex > 0.1 THEN
  IF g_batches[i_blocked_unit].cur_stage = i_blocked_stage THEN
    cap := 0.9;
  ELSE
    cap := 0.5;
  END_IF;
  amount := prev_flex * cap;
  IF amount > remain THEN amount := remain; END_IF;

  g_schedule[i_blocked_unit].stages[i_blocked_stage].calc_time :=
    g_schedule[i_blocked_unit].stages[i_blocked_stage].calc_time + amount;
  g_schedule[i_blocked_unit].stages[i_blocked_stage].exit_time :=
    g_schedule[i_blocked_unit].stages[i_blocked_stage].exit_time + amount;
  sc := g_schedule[i_blocked_unit].stage_count;
  FOR si := i_blocked_stage + 1 TO sc DO
    g_schedule[i_blocked_unit].stages[si].entry_time :=
      g_schedule[i_blocked_unit].stages[si].entry_time + amount;
    g_schedule[i_blocked_unit].stages[si].exit_time :=
      g_schedule[i_blocked_unit].stages[si].exit_time + amount;
  END_FOR;

  FOR qi := 1 TO 3 DO
    FOR si := 1 TO g_tasks[qi].count DO
      IF g_tasks[qi].queue[si].unit = i_blocked_unit
         AND g_tasks[qi].queue[si].stage >= i_blocked_stage THEN
        g_tasks[qi].queue[si].start_time :=
          g_tasks[qi].queue[si].start_time + amount;
        g_tasks[qi].queue[si].finish_time :=
          g_tasks[qi].queue[si].finish_time + amount;
      END_IF;
    END_FOR;
  END_FOR;

  remain := remain - amount;
  o_total_delay := o_total_delay + amount;
END_IF;

IF remain <= 0.1 THEN
  o_solved := TRUE;
END_IF;

(* If not solved, partial resolution was still applied *)
          
END_FUNCTION_BLOCK

FUNCTION_BLOCK TSK_FB_Scheduler
  VAR_INPUT
    i_run : BOOL;
    i_time_s : REAL;
  END_VAR
  VAR_OUTPUT
    o_phase : INT;
    o_batch_cnt : INT;
    o_task_cnt : INT;
    o_cycle_cnt : INT;
    o_conflict : BOOL;
  END_VAR
  VAR_EXTERNAL
    g_batches : ARRAY[1..10] OF BATCH_T;
    g_units : ARRAY[1..10] OF UNIT_T;
    g_programs : ARRAY[1..10] OF TREATMENT_PROGRAM_T;
    g_tasks : ARRAY[1..3] OF TSK_QUEUE_T;
    g_schedule : ARRAY[1..10] OF TSK_SCHEDULE_T;
    g_dep_pending : DEP_PENDING_WRITE_T;
  END_VAR
  VAR
    phase : INT := 0;
    next_phase : INT;
    batch_idx : INT;
    batch_list : ARRAY[1..10] OF INT;
    batch_count : INT;
    conflict_iter : INT;
    MAX_CONFLICT_ITER : INT := 20;
    fb_calc : TSK_FB_CalcSchedule;
    fb_create : TSK_FB_CreateTasks;
    fb_swap : TSK_FB_SwapTasks;
    fb_analyze : TSK_FB_Analyze;
    fb_resolve : TSK_FB_Resolve;
    fb_notrt : TSK_FB_NoTreatment;
    fb_find : STC_FB_FindTransporter;
    sched_trans : INT;
    bi : INT;
    ti : INT;
    qi : INT;
    ui : INT;
    total_tasks : INT;
    ins_i : INT;
    ins_j : INT;
    ins_cnt : INT;
    tmp_task : TSK_TASK_T;
    cycle_count : INT := 0;
  END_VAR

            IF NOT i_run THEN
  phase := 0;
  o_phase := 0;
  RETURN;
END_IF;

next_phase := phase;

(* ══════════════════════════════════════════════════════════════ *)
(* PHASE 0: STOPPED — wait for i_run                            *)
(* ══════════════════════════════════════════════════════════════ *)
IF phase = 0 THEN
  next_phase := 1;

(* ══════════════════════════════════════════════════════════════ *)
(* PHASE 1: INIT — collect active batches                       *)
(* ══════════════════════════════════════════════════════════════ *)
ELSIF phase = 1 THEN
  batch_count := 0;
  FOR bi := 1 TO 10 DO
    (* Active batch: state = IN_PROCESS (1) or has valid program *)
    IF g_batches[bi].state = 1 THEN
      batch_count := batch_count + 1;
      batch_list[batch_count] := bi;
    END_IF;
  END_FOR;
  o_batch_cnt := batch_count;
  conflict_iter := 0;

  IF batch_count = 0 THEN
    (* No active batches — go to READY directly *)
    next_phase := 10000;
  ELSE
    next_phase := 1000;
  END_IF;

(* ══════════════════════════════════════════════════════════════ *)
(* PHASE 1000: SCHEDULE_START                                   *)
(* ══════════════════════════════════════════════════════════════ *)
ELSIF phase = 1000 THEN
  batch_idx := 1;
  next_phase := 1001;

(* ══════════════════════════════════════════════════════════════ *)
(* PHASE 1001..1010: SCHEDULE per batch (one per tick)          *)
(* ══════════════════════════════════════════════════════════════ *)
ELSIF phase >= 1001 AND phase <= 1010 THEN
  IF batch_idx <= batch_count THEN
    ui := batch_list[batch_idx];

    (* Find transporter for this unit — first one with matching task_area *)
    fb_find(i_lift_stn := g_units[ui].location, i_sink_stn := 0);
    sched_trans := fb_find.o_trans_id;
    IF sched_trans = 0 THEN sched_trans := 1; END_IF;  (* fallback default *)

    fb_calc(i_unit := ui, i_trans := sched_trans, i_time_s := i_time_s);

    batch_idx := batch_idx + 1;
    IF batch_idx <= batch_count THEN
      next_phase := phase + 1;
    ELSE
      next_phase := 1900;
    END_IF;
  ELSE
    next_phase := 1900;
  END_IF;

(* ══════════════════════════════════════════════════════════════ *)
(* PHASE 1900: SCHEDULE_DONE                                    *)
(* ══════════════════════════════════════════════════════════════ *)
ELSIF phase = 1900 THEN
  next_phase := 2000;

(* ══════════════════════════════════════════════════════════════ *)
(* PHASE 2000: TASKS_START — clear all task queues              *)
(* ══════════════════════════════════════════════════════════════ *)
ELSIF phase = 2000 THEN
  FOR ti := 1 TO 3 DO
    g_tasks[ti].count := 0;
    FOR qi := 1 TO 10 DO
      g_tasks[ti].queue[qi].unit := 0;
      g_tasks[ti].queue[qi].stage := 0;
      g_tasks[ti].queue[qi].lift_station := 0;
      g_tasks[ti].queue[qi].sink_station := 0;
      g_tasks[ti].queue[qi].start_time := 0.0;
      g_tasks[ti].queue[qi].finish_time := 0.0;
      g_tasks[ti].queue[qi].calc_time := 0.0;
      g_tasks[ti].queue[qi].min_time := 0.0;
      g_tasks[ti].queue[qi].max_time := 0.0;
    END_FOR;
  END_FOR;
  batch_idx := 1;
  next_phase := 2001;

(* ══════════════════════════════════════════════════════════════ *)
(* PHASE 2001..2010: CREATE_TASKS per batch (one per tick)      *)
(* ══════════════════════════════════════════════════════════════ *)
ELSIF phase >= 2001 AND phase <= 2010 THEN
  IF batch_idx <= batch_count THEN
    ui := batch_list[batch_idx];
    fb_create(i_unit := ui);
    batch_idx := batch_idx + 1;
    IF batch_idx <= batch_count THEN
      next_phase := phase + 1;
    ELSE
      next_phase := 2200;
    END_IF;
  ELSE
    next_phase := 2200;
  END_IF;

(* ══════════════════════════════════════════════════════════════ *)
(* PHASE 2200: TASKS_SORT — insertion sort each queue by time   *)
(* ══════════════════════════════════════════════════════════════ *)
ELSIF phase = 2200 THEN
  FOR ti := 1 TO 3 DO
    ins_cnt := g_tasks[ti].count;
    IF ins_cnt >= 2 THEN
      FOR ins_i := 2 TO ins_cnt DO
        tmp_task := g_tasks[ti].queue[ins_i];
        ins_j := ins_i - 1;
        WHILE ins_j >= 1 AND g_tasks[ti].queue[ins_j].start_time > tmp_task.start_time DO
          g_tasks[ti].queue[ins_j + 1] := g_tasks[ti].queue[ins_j];
          ins_j := ins_j - 1;
        END_WHILE;
        g_tasks[ti].queue[ins_j + 1] := tmp_task;
      END_FOR;
    END_IF;
  END_FOR;
  next_phase := 2201;

(* ══════════════════════════════════════════════════════════════ *)
(* PHASE 2201: TASKS_SWAP                                       *)
(* ══════════════════════════════════════════════════════════════ *)
ELSIF phase = 2201 THEN
  fb_swap();
  next_phase := 2202;

(* ══════════════════════════════════════════════════════════════ *)
(* PHASE 2202: TASKS_ANALYZE                                    *)
(* ══════════════════════════════════════════════════════════════ *)
ELSIF phase = 2202 THEN
  fb_analyze();
  o_conflict := fb_analyze.o_has_conflict;
  IF fb_analyze.o_has_conflict THEN
    next_phase := 2203;
  ELSE
    next_phase := 2204;
  END_IF;

(* ══════════════════════════════════════════════════════════════ *)
(* PHASE 2203: TASKS_RESOLVE                                    *)
(* One conflict per cycle → recalculate                         *)
(* ══════════════════════════════════════════════════════════════ *)
ELSIF phase = 2203 THEN
  fb_resolve(
    i_conf_unit     := fb_analyze.o_conf_unit,
    i_conf_stage    := fb_analyze.o_conf_stage,
    i_conf_trans    := fb_analyze.o_conf_trans,
    i_blocked_unit  := fb_analyze.o_blocked_unit,
    i_blocked_stage := fb_analyze.o_blocked_stage,
    i_deficit       := fb_analyze.o_deficit
  );

  conflict_iter := conflict_iter + 1;

  IF conflict_iter >= MAX_CONFLICT_ITER THEN
    (* Max iterations reached — accept partial solution *)
    next_phase := 2204;
  ELSE
    (* Re-analyze: SORT → SWAP → ANALYZE again *)
    next_phase := 2200;
  END_IF;

(* ══════════════════════════════════════════════════════════════ *)
(* PHASE 2204: TASKS_NO_TREATMENT                               *)
(* Task list is stable (no conflicts). Create unit-target tasks *)
(* ══════════════════════════════════════════════════════════════ *)
ELSIF phase = 2204 THEN
  fb_notrt(i_time_s := i_time_s);
  o_conflict := FALSE;
  next_phase := 10000;

(* ══════════════════════════════════════════════════════════════ *)
(* PHASE 10000: READY — cycle complete                          *)
(* ══════════════════════════════════════════════════════════════ *)
ELSIF phase = 10000 THEN
  (* Count total tasks *)
  total_tasks := 0;
  FOR ti := 1 TO 3 DO
    total_tasks := total_tasks + g_tasks[ti].count;
  END_FOR;
  o_task_cnt := total_tasks;
  next_phase := 10100;

(* ══════════════════════════════════════════════════════════════ *)
(* PHASE 10100: CHECK_DEP_PENDING — DEP activated a batch       *)
(* Copy pending data to globals and trigger full recalculation  *)
(* ══════════════════════════════════════════════════════════════ *)
ELSIF phase = 10100 THEN
  IF g_dep_pending.valid THEN
    (* Apply DEP’s pending data: programs + stage change *)
    FOR ui := 1 TO 10 DO
      g_programs[ui] := g_dep_pending.programs[ui];
    END_FOR;
    IF g_dep_pending.batch_unit >= 1 AND g_dep_pending.batch_unit <= 10 THEN
      g_batches[g_dep_pending.batch_unit].cur_stage := g_dep_pending.batch_stage;
    END_IF;
    g_dep_pending.valid := FALSE;
    (* Full recalculation with new data *)
    next_phase := 1;
  ELSE
    next_phase := 10110;
  END_IF;

(* ══════════════════════════════════════════════════════════════ *)
(* PHASE 10110: RESTART — begin new cycle                       *)
(* ══════════════════════════════════════════════════════════════ *)
ELSIF phase = 10110 THEN
  cycle_count := cycle_count + 1;
  o_cycle_cnt := cycle_count;
  next_phase := 1;  (* back to INIT *)

(* ══════════════════════════════════════════════════════════════ *)
(* Unknown phase → reset to INIT                                *)
(* ══════════════════════════════════════════════════════════════ *)
ELSE
  next_phase := 1;
END_IF;

(* ── Phase assignment at end of scan ── *)
phase := next_phase;
o_phase := phase;
          
END_FUNCTION_BLOCK

FUNCTION_BLOCK TWA_FB_CalcLimits
  VAR_EXTERNAL
    MAX_TRANSPORTERS : INT;
    AVOID_PASS : INT;
    AVOID_BLOCK : INT;
    MIN_WORK_AREA : REAL;
  END_VAR
  VAR
    i : INT;
    j : INT;
    k : INT;
    stn_num : INT;
    stn_x : REAL;
    avoid_st : INT;
    min_x : REAL;
    max_x : REAL;
    current_x : REAL;
    avoid_dist : REAL;
    is_target : BOOL;
    new_val : REAL;
    left_s2_x : REAL;
    right_s2_x : REAL;
    has_left_s2 : BOOL;
    has_right_s2 : BOOL;
    midpoint : REAL;
    n_active : INT;
    w_idx : ARRAY[1..3] OF INT;
    w_xpos : ARRAY[1..3] OF REAL;
    w_phase : ARRAY[1..3] OF INT;
    w_target : ARRAY[1..3] OF REAL;
    w_avoid : ARRAY[1..3] OF REAL;
    w_can_evade : ARRAY[1..3] OF BOOL;
    w_priority : ARRAY[1..3] OF REAL;
    min_idx : INT;
    tmp_int : INT;
    tmp_real : REAL;
    tmp_bool : BOOL;
    a_wins : BOOL;
    restrict_x : REAL;
    between : INT;
    chain_ofs : REAL;
    cur_min : REAL;
    cur_max : REAL;
    adjusted : REAL;
    left_right : BOOL;
    right_right : BOOL;
    left_left : BOOL;
    right_left : BOOL;
    safety_val : REAL;
    work_area : REAL;
    other_x : REAL;
    other_avoid : REAL;
  END_VAR

            (* ================================================================
   PHASE 1: Station-based restrictions from g_avoid_status
   For each active transporter, search stations near current_station
   and restrict x_min/x_max based on avoid_status 1 (pass) and 2 (block).
   ================================================================ *)
FOR i := 1 TO MAX_TRANSPORTERS DO
  IF NOT g_state[i].active THEN
    CONTINUE;
  END_IF;

  min_x := g_cfg[i].x_min_limit;
  max_x := g_cfg[i].x_max_limit;
  current_x := g_state[i].x_mm;
  avoid_dist := g_cfg[i].x_avoid_mm;

  (* If no limits configured, lock to current position *)
  IF (min_x < 1.0) OR (max_x < 1.0) THEN
    g_state[i].x_min_limit := current_x;
    g_state[i].x_max_limit := current_x;
    CONTINUE;
  END_IF;

  has_left_s2 := FALSE;
  has_right_s2 := FALSE;
  left_s2_x := 0.0;
  right_s2_x := 0.0;

  (* --- Search downward (smaller station numbers) from current_station --- *)
  stn_num := g_state[i].current_station - 1;
  WHILE stn_num >= 101 DO
    IF g_stations[stn_num].tank_id = 0 THEN
      stn_num := stn_num - 1;
      CONTINUE;
    END_IF;

    stn_x := g_stations[stn_num].x_position;
    IF stn_x < min_x THEN
      EXIT;
    END_IF;

    avoid_st := g_avoid_status[stn_num];

    (* AVOID_PASS: passable unless it is this transporter's target station *)
    IF avoid_st = AVOID_PASS THEN
      is_target := (stn_num = g_state[i].lift_station_target)
               OR  (stn_num = g_state[i].sink_station_target);
      IF is_target THEN
        IF current_x < stn_x THEN
          new_val := stn_x - avoid_dist;
          IF new_val < max_x THEN max_x := new_val; END_IF;
          right_s2_x := stn_x;
          has_right_s2 := TRUE;
        ELSE
          new_val := stn_x + avoid_dist;
          IF new_val > min_x THEN min_x := new_val; END_IF;
          left_s2_x := stn_x;
          has_left_s2 := TRUE;
        END_IF;
        EXIT;
      END_IF;
      (* else: passable, keep searching *)
    END_IF;

    (* AVOID_BLOCK: hard block — transporter cannot cross *)
    IF avoid_st = AVOID_BLOCK THEN
      IF current_x < stn_x THEN
        new_val := stn_x - avoid_dist;
        IF new_val < max_x THEN max_x := new_val; END_IF;
        right_s2_x := stn_x;
        has_right_s2 := TRUE;
      ELSE
        new_val := stn_x + avoid_dist;
        IF new_val > min_x THEN min_x := new_val; END_IF;
        left_s2_x := stn_x;
        has_left_s2 := TRUE;
      END_IF;
      EXIT;
    END_IF;

    stn_num := stn_num - 1;
  END_WHILE;

  (* --- Search upward (larger station numbers) from current_station --- *)
  stn_num := g_state[i].current_station + 1;
  WHILE stn_num <= 125 DO
    IF g_stations[stn_num].tank_id = 0 THEN
      stn_num := stn_num + 1;
      CONTINUE;
    END_IF;

    stn_x := g_stations[stn_num].x_position;
    IF stn_x > max_x THEN
      EXIT;
    END_IF;

    avoid_st := g_avoid_status[stn_num];

    IF avoid_st = AVOID_PASS THEN
      is_target := (stn_num = g_state[i].lift_station_target)
               OR  (stn_num = g_state[i].sink_station_target);
      IF is_target THEN
        IF current_x < stn_x THEN
          new_val := stn_x - avoid_dist;
          IF new_val < max_x THEN max_x := new_val; END_IF;
          right_s2_x := stn_x;
          has_right_s2 := TRUE;
        ELSE
          new_val := stn_x + avoid_dist;
          IF new_val > min_x THEN min_x := new_val; END_IF;
          left_s2_x := stn_x;
          has_left_s2 := TRUE;
        END_IF;
        EXIT;
      END_IF;
    END_IF;

    IF avoid_st = AVOID_BLOCK THEN
      IF current_x < stn_x THEN
        new_val := stn_x - avoid_dist;
        IF new_val < max_x THEN max_x := new_val; END_IF;
        right_s2_x := stn_x;
        has_right_s2 := TRUE;
      ELSE
        new_val := stn_x + avoid_dist;
        IF new_val > min_x THEN min_x := new_val; END_IF;
        left_s2_x := stn_x;
        has_left_s2 := TRUE;
      END_IF;
      EXIT;
    END_IF;

    stn_num := stn_num + 1;
  END_WHILE;

  (* Conflict resolution: trapped between two BLOCK stations *)
  IF (min_x >= max_x) AND has_left_s2 AND has_right_s2 THEN
    midpoint := (left_s2_x + right_s2_x) / 2.0;
    min_x := midpoint - 5.0;
    max_x := midpoint + 5.0;
  END_IF;

  g_state[i].x_min_limit := min_x;
  g_state[i].x_max_limit := max_x;
END_FOR;

(* ================================================================
   STEP 2.0: Basic safety distance — current positions
   Every active transporter pushes neighbors away by x_avoid_mm.
   ================================================================ *)
FOR i := 1 TO MAX_TRANSPORTERS DO
  IF NOT g_state[i].active THEN
    CONTINUE;
  END_IF;

  current_x := g_state[i].x_mm;
  avoid_dist := g_cfg[i].x_avoid_mm;

  FOR j := 1 TO MAX_TRANSPORTERS DO
    IF j = i THEN CONTINUE; END_IF;
    IF NOT g_state[j].active THEN CONTINUE; END_IF;

    other_x := g_state[j].x_mm;

    IF other_x > current_x THEN
      (* j is to the RIGHT of i — restrict j's x_min *)
      new_val := current_x + avoid_dist;
      IF new_val > g_state[j].x_min_limit THEN
        g_state[j].x_min_limit := new_val;
      END_IF;
    ELSIF other_x < current_x THEN
      (* j is to the LEFT of i — restrict j's x_max *)
      new_val := current_x - avoid_dist;
      IF new_val < g_state[j].x_max_limit THEN
        g_state[j].x_max_limit := new_val;
      END_IF;
    END_IF;
  END_FOR;
END_FOR;

(* ================================================================
   STEP 2.2: Priority-based collision avoidance
   ================================================================ *)

(* --- 2.2.1: Build sorted array of active transporters by x-position --- *)
n_active := 0;
FOR i := 1 TO MAX_TRANSPORTERS DO
  IF g_state[i].active THEN
    n_active := n_active + 1;
    w_idx[n_active] := i;
    w_xpos[n_active] := g_state[i].x_mm;
    w_phase[n_active] := g_state[i].phase;
    w_target[n_active] := g_state[i].target_x;
    w_avoid[n_active] := g_cfg[i].x_avoid_mm;
  END_IF;
END_FOR;

(* Selection sort by x-position (ascending) *)
FOR i := 1 TO n_active - 1 DO
  min_idx := i;
  FOR j := i + 1 TO n_active DO
    IF w_xpos[j] < w_xpos[min_idx] THEN
      min_idx := j;
    END_IF;
  END_FOR;
  IF min_idx <> i THEN
    tmp_int := w_idx[i];    w_idx[i] := w_idx[min_idx];    w_idx[min_idx] := tmp_int;
    tmp_real := w_xpos[i];  w_xpos[i] := w_xpos[min_idx];  w_xpos[min_idx] := tmp_real;
    tmp_int := w_phase[i];  w_phase[i] := w_phase[min_idx]; w_phase[min_idx] := tmp_int;
    tmp_real := w_target[i]; w_target[i] := w_target[min_idx]; w_target[min_idx] := tmp_real;
    tmp_real := w_avoid[i];  w_avoid[i] := w_avoid[min_idx];  w_avoid[min_idx] := tmp_real;
  END_IF;
END_FOR;

(* --- 2.2.2: Calculate canEvade and priority --- *)
FOR i := 1 TO n_active DO
  k := w_idx[i];

  (* canEvade rules:
     - phase 2 or 4 (Z-movement): cannot evade
     - working area too small: cannot evade *)
  w_can_evade[i] := TRUE;
  IF (w_phase[i] = 2) OR (w_phase[i] = 4) THEN
    w_can_evade[i] := FALSE;
  END_IF;
  work_area := g_state[k].x_max_limit - g_state[k].x_min_limit;
  IF work_area < MIN_WORK_AREA THEN
    w_can_evade[i] := FALSE;
  END_IF;

  w_priority[i] := TWA_CalcPriority(
    i_phase := w_phase[i],
    i_can_evade := w_can_evade[i],
    i_x_pos := w_xpos[i],
    i_x_target := w_target[i]
  );
END_FOR;

(* Skip Steps 2.2.3-2.2.5 if fewer than 2 active transporters *)
IF n_active >= 2 THEN

  (* --- 2.2.3: Priority restrictions (higher priority → lower priority) --- *)
  FOR i := 1 TO n_active DO
    (* Skip idle transporters — they don't set priority restrictions *)
    IF w_phase[i] = 0 THEN CONTINUE; END_IF;

    FOR j := 1 TO n_active DO
      IF i = j THEN CONTINUE; END_IF;

      (* Determine if i has higher priority than j *)
      a_wins := FALSE;
      IF w_priority[i] > w_priority[j] THEN
        a_wins := TRUE;
      ELSIF (w_priority[i] = w_priority[j]) AND (w_idx[i] < w_idx[j]) THEN
        a_wins := TRUE;
      END_IF;

      IF NOT a_wins THEN CONTINUE; END_IF;

      (* Higher priority transporter uses target for phase 1/3, else current pos *)
      IF (w_phase[i] = 1) OR (w_phase[i] = 3) THEN
        restrict_x := w_target[i];
      ELSE
        restrict_x := w_xpos[i];
      END_IF;

      k := w_idx[j];
      cur_min := g_state[k].x_min_limit;
      cur_max := g_state[k].x_max_limit;

      IF w_xpos[i] < w_xpos[j] THEN
        (* i is LEFT, j is RIGHT — i sets j's x_min *)
        between := j - i - 1;
        chain_ofs := w_avoid[i] + INT_TO_REAL(between) * (MIN_WORK_AREA + w_avoid[i]);
        new_val := restrict_x + chain_ofs;

        IF new_val > cur_min THEN
          IF new_val <= (cur_max - MIN_WORK_AREA) THEN
            g_state[k].x_min_limit := new_val;
          ELSE
            adjusted := cur_max - MIN_WORK_AREA;
            IF adjusted > cur_min THEN
              g_state[k].x_min_limit := adjusted;
            END_IF;
          END_IF;
        END_IF;

      ELSIF w_xpos[i] > w_xpos[j] THEN
        (* i is RIGHT, j is LEFT — i sets j's x_max *)
        between := i - j - 1;
        chain_ofs := w_avoid[i] + INT_TO_REAL(between) * (MIN_WORK_AREA + w_avoid[i]);
        new_val := restrict_x - chain_ofs;

        IF new_val < cur_max THEN
          IF new_val >= (cur_min + MIN_WORK_AREA) THEN
            g_state[k].x_max_limit := new_val;
          ELSE
            adjusted := cur_min + MIN_WORK_AREA;
            IF adjusted < cur_max THEN
              g_state[k].x_max_limit := adjusted;
            END_IF;
          END_IF;
        END_IF;
      END_IF;
    END_FOR;
  END_FOR;

  (* --- 2.2.4: Bidirectional safety (both moving same direction) --- *)
  FOR i := 1 TO n_active - 1 DO
    j := i + 1;
    (* i = left (smaller x), j = right (larger x) — sorted array *)

    left_right := ((w_phase[i] = 1) OR (w_phase[i] = 3)) AND (w_target[i] > w_xpos[i]);
    right_right := ((w_phase[j] = 1) OR (w_phase[j] = 3)) AND (w_target[j] > w_xpos[j]);
    left_left := ((w_phase[i] = 1) OR (w_phase[i] = 3)) AND (w_target[i] < w_xpos[i]);
    right_left := ((w_phase[j] = 1) OR (w_phase[j] = 3)) AND (w_target[j] < w_xpos[j]);

    IF left_right AND right_right THEN
      (* Both moving right — left chasing right *)
      safety_val := w_xpos[i] + w_avoid[i];
      k := w_idx[j];
      IF safety_val > g_state[k].x_min_limit THEN
        g_state[k].x_min_limit := safety_val;
      END_IF;
    END_IF;

    IF left_left AND right_left THEN
      (* Both moving left — right chasing left *)
      safety_val := w_xpos[j] - w_avoid[j];
      k := w_idx[i];
      IF safety_val < g_state[k].x_max_limit THEN
        g_state[k].x_max_limit := safety_val;
      END_IF;
    END_IF;
  END_FOR;

  (* --- 2.2.5: Validate limits (trap detection) --- *)
  FOR i := 1 TO n_active DO
    k := w_idx[i];
    IF g_state[k].x_min_limit > g_state[k].x_max_limit THEN
      (* Trapped — lock in place *)
      g_state[k].x_min_limit := g_state[k].x_mm;
      g_state[k].x_max_limit := g_state[k].x_mm;
    END_IF;
  END_FOR;

END_IF;  (* n_active >= 2 *)
          
END_FUNCTION_BLOCK

FUNCTION_BLOCK FB_ClearConfig
  VAR_EXTERNAL
    g_station_count : INT;
    g_stations : ARRAY[101..125] OF STATION_T;
    g_cfg : ARRAY[1..3] OF TRANSPORTER_CFG_T;
    g_state : ARRAY[1..3] OF TRANSPORTER_STATE_T;
    g_cmd_start : ARRAY[1..3] OF BOOL;
    g_cmd_lift_station : ARRAY[1..3] OF INT;
    g_cmd_sink_station : ARRAY[1..3] OF INT;
    g_units : ARRAY[1..10] OF UNIT_T;
    g_batches : ARRAY[1..10] OF BATCH_T;
    g_programs : ARRAY[1..10] OF TREATMENT_PROGRAM_T;
    g_avoid_status : ARRAY[101..125] OF INT;
  END_VAR
  VAR
    i : INT;
    j : INT;
    k : INT;
  END_VAR

            (* --- Clear all stations --- *)
FOR i := 101 TO 125 DO
  g_stations[i].tank_id       := 0;
  g_stations[i].status        := 0;
  g_stations[i].x_position    := 0.0;
  g_stations[i].y_position    := 0.0;
  g_stations[i].z_position    := 0.0;
  g_stations[i].stn_type      := 0;
  g_stations[i].dropping_time := 0.0;
  g_stations[i].device_delay  := 0.0;
END_FOR;
g_station_count := 0;

(* --- Clear all transporter configs --- *)
FOR i := 1 TO 3 DO
  g_cfg[i].x_min_limit   := 0.0;
  g_cfg[i].x_max_limit   := 0.0;
  g_cfg[i].y_min_limit   := 0.0;
  g_cfg[i].y_max_limit   := 0.0;
  g_cfg[i].x_avoid_mm    := 0.0;
  g_cfg[i].y_avoid_mm    := 0.0;
  g_cfg[i].phys2d.x_accel_s     := 0.0;
  g_cfg[i].phys2d.x_decel_s     := 0.0;
  g_cfg[i].phys2d.x_max_mm_s    := 0.0;
  g_cfg[i].phys2d.z_total_mm    := 0.0;
  g_cfg[i].phys2d.z_slow_dry_mm := 0.0;
  g_cfg[i].phys2d.z_slow_wet_mm := 0.0;
  g_cfg[i].phys2d.z_slow_end_mm := 0.0;
  g_cfg[i].phys2d.z_slow_mm_s   := 0.0;
  g_cfg[i].phys2d.z_fast_mm_s   := 0.0;
  g_cfg[i].phys2d.drip_delay_s  := 0.0;
  g_cfg[i].phys2d.avoid_mm      := 0.0;
  FOR j := 1 TO 4 DO
    g_cfg[i].task_area[j].min_lift := 0;
    g_cfg[i].task_area[j].max_lift := 0;
    g_cfg[i].task_area[j].min_sink := 0;
    g_cfg[i].task_area[j].max_sink := 0;
  END_FOR;
END_FOR;

(* --- Clear avoid status --- *)
FOR i := 101 TO 125 DO
  g_avoid_status[i] := 0;
END_FOR;

(* --- Clear all transporter states --- *)
FOR i := 1 TO 3 DO
  g_state[i].active              := FALSE;
  g_state[i].phase               := 0;
  g_state[i].z_stage             := 0;
  g_state[i].x_mm                := 0.0;
  g_state[i].z_mm                := 0.0;
  g_state[i].vel_x               := 0.0;
  g_state[i].vel_z               := 0.0;
  g_state[i].current_station     := 0;
  g_state[i].lift_station_target := 0;
  g_state[i].sink_station_target := 0;
  g_state[i].target_x            := 0.0;
  g_state[i].x_min_limit         := 0.0;
  g_state[i].x_max_limit         := 0.0;
  g_state[i].z_timer_s           := 0.0;
  g_cmd_start[i]        := FALSE;
  g_cmd_lift_station[i]  := 0;
  g_cmd_sink_station[i]  := 0;
END_FOR;

(* --- Clear all units --- *)
FOR i := 1 TO 10 DO
  g_units[i].location := 0;
  g_units[i].status   := 0;
  g_units[i].state    := 0;
  g_units[i].target   := 0;
END_FOR;

(* --- Clear all batches --- *)
FOR i := 1 TO 10 DO
  g_batches[i].batch_code := 0;
  g_batches[i].state      := 0;
  g_batches[i].prog_id    := 0;
  g_batches[i].cur_stage      := 0;
END_FOR;

(* --- Clear all treatment programs --- *)
FOR i := 1 TO 10 DO
  g_programs[i].program_id := 0;
  FOR j := 1 TO 30 DO
    FOR k := 1 TO 5 DO
      g_programs[i].stages[j].stations[k] := 0;
    END_FOR;
    g_programs[i].stages[j].min_time := 0;
    g_programs[i].stages[j].max_time := 0;
    g_programs[i].stages[j].cal_time := 0;
  END_FOR;
END_FOR;
          
END_FUNCTION_BLOCK

PROGRAM PLC_PRG
  VAR_EXTERNAL
    g_station_count : INT;
    g_stations : ARRAY[101..125] OF STATION_T;
    g_cfg : ARRAY[1..3] OF TRANSPORTER_CFG_T;
    g_state : ARRAY[1..3] OF TRANSPORTER_STATE_T;
    g_cmd_start : ARRAY[1..3] OF BOOL;
    g_cmd_lift_station : ARRAY[1..3] OF INT;
    g_cmd_sink_station : ARRAY[1..3] OF INT;
    qw_t1_x_mm : INT;
    qw_t1_z_mm : INT;
    qw_t1_vel_x10 : INT;
    qw_t1_phase : INT;
    qw_t1_z_stage : INT;
    qw_t1_cur_st : INT;
    qw_t1_lift_tgt : INT;
    qw_t1_sink_tgt : INT;
    qw_t1_active : INT;
    qw_t2_x_mm : INT;
    qw_t2_z_mm : INT;
    qw_t2_vel_x10 : INT;
    qw_t2_phase : INT;
    qw_t2_z_stage : INT;
    qw_t2_cur_st : INT;
    qw_t2_lift_tgt : INT;
    qw_t2_sink_tgt : INT;
    qw_t2_active : INT;
    qw_station_cnt : INT;
    qw_init_done : INT;
    qw_cycle_cnt : INT;
    iw_cmd_start_1 : INT;
    iw_cmd_lift_1 : INT;
    iw_cmd_sink_1 : INT;
    iw_cmd_start_2 : INT;
    iw_cmd_lift_2 : INT;
    iw_cmd_sink_2 : INT;
    iw_cfg_seq : INT;
    iw_cfg_cmd : INT;
    iw_cfg_param : INT;
    iw_cfg_d0 : INT;
    iw_cfg_d1 : INT;
    iw_cfg_d2 : INT;
    iw_cfg_d3 : INT;
    iw_cfg_d4 : INT;
    iw_cfg_d5 : INT;
    iw_cfg_d6 : INT;
    qw_cfg_ack : INT;
    g_units : ARRAY[1..10] OF UNIT_T;
    qw_u1_loc : INT;
    qw_u1_status : INT;
    qw_u1_state : INT;
    qw_u1_target : INT;
    qw_u2_loc : INT;
    qw_u2_status : INT;
    qw_u2_state : INT;
    qw_u2_target : INT;
    qw_u3_loc : INT;
    qw_u3_status : INT;
    qw_u3_state : INT;
    qw_u3_target : INT;
    qw_u4_loc : INT;
    qw_u4_status : INT;
    qw_u4_state : INT;
    qw_u4_target : INT;
    qw_u5_loc : INT;
    qw_u5_status : INT;
    qw_u5_state : INT;
    qw_u5_target : INT;
    qw_u6_loc : INT;
    qw_u6_status : INT;
    qw_u6_state : INT;
    qw_u6_target : INT;
    qw_u7_loc : INT;
    qw_u7_status : INT;
    qw_u7_state : INT;
    qw_u7_target : INT;
    qw_u8_loc : INT;
    qw_u8_status : INT;
    qw_u8_state : INT;
    qw_u8_target : INT;
    qw_u9_loc : INT;
    qw_u9_status : INT;
    qw_u9_state : INT;
    qw_u9_target : INT;
    qw_u10_loc : INT;
    qw_u10_status : INT;
    qw_u10_state : INT;
    qw_u10_target : INT;
    qw_unit_ack : INT;
    qw_b1_code : INT;
    qw_b2_code : INT;
    qw_b3_code : INT;
    qw_b4_code : INT;
    qw_b5_code : INT;
    qw_b6_code : INT;
    qw_b7_code : INT;
    qw_b8_code : INT;
    qw_b9_code : INT;
    qw_b10_code : INT;
    iw_unit_seq : INT;
    iw_unit_id : INT;
    iw_unit_loc : INT;
    iw_unit_status : INT;
    iw_unit_state : INT;
    iw_unit_target : INT;
    g_batches : ARRAY[1..10] OF BATCH_T;
    g_programs : ARRAY[1..10] OF TREATMENT_PROGRAM_T;
    g_avoid_status : ARRAY[101..125] OF INT;
    iw_batch_seq : INT;
    iw_batch_unit : INT;
    iw_batch_code : INT;
    iw_batch_state : INT;
    iw_batch_prog_id : INT;
    qw_batch_ack : INT;
    iw_prog_seq : INT;
    iw_prog_unit : INT;
    iw_prog_stage : INT;
    iw_prog_s1 : INT;
    iw_prog_s2 : INT;
    iw_prog_s3 : INT;
    iw_prog_s4 : INT;
    iw_prog_s5 : INT;
    iw_prog_min_time : INT;
    iw_prog_max_time : INT;
    iw_prog_cal_time : INT;
    qw_prog_ack : INT;
    g_epoch_h : INT;
    g_time_s : REAL;
    iw_epoch_h : INT;
    iw_time_hi : INT;
    iw_time_lo : INT;
    g_schedule : ARRAY[1..10] OF TSK_SCHEDULE_T;
    g_tasks : ARRAY[1..3] OF TSK_QUEUE_T;
    g_dep_stable : BOOL;
  END_VAR
  VAR
    init_done : BOOL := FALSE;
    last_cfg_seq : INT := 0;
    last_unit_seq : INT := 0;
    last_batch_seq : INT := 0;
    last_prog_seq : INT := 0;
    j : INT;
    k : INT;
    i : INT;
    stn_num : INT;
    idx : INT;
    station_type : INT;
    device_delay : REAL;
    drop_time : REAL;
    arrived_x : BOOL;
    nearest_num : INT;
    min_dist : REAL;
    dx : REAL;
    tmp_x : REAL;
    tmp_vx : REAL;
    fb_x1 : SIM_FB_XMotion;
    fb_x2 : SIM_FB_XMotion;
    fb_x3 : SIM_FB_XMotion;
    fb_z1 : SIM_FB_ZMotion;
    fb_z2 : SIM_FB_ZMotion;
    fb_z3 : SIM_FB_ZMotion;
    twa_calc : TWA_FB_CalcLimits;
    lookup : STC_FB_FindStation;
    clear_cfg : FB_ClearConfig;
    cycle_count : INT;
    tmp_z : REAL;
    tmp_zs : INT;
    tmp_zt : REAL;
    arrived_z : BOOL;
    tsk_sched : TSK_FB_Scheduler;
    dep_sched : DEP_FB_Scheduler;
  END_VAR

            (* ============================================================
   CONFIG UPLOAD HANDLER
   Gateway writes station data one at a time via Modbus IW regs.
   Sequence number change triggers processing.
   cmd=1: write_station  cmd=2: init  cmd=3: clear_all
   ============================================================ *)
IF iw_cfg_seq <> last_cfg_seq THEN
  last_cfg_seq := iw_cfg_seq;

  IF iw_cfg_cmd = 3 THEN
    (* --- Clear all config data --- *)
    clear_cfg();
    init_done := FALSE;
    qw_init_done := 0;
    qw_station_cnt := 0;
    qw_cfg_ack := iw_cfg_seq;

